18:	FB_FileClose_Indo.bExecute:=TRUE;
	 IF NOT FB_FileClose_Indo.bBusy AND NOT FB_FileClose_Indo.bError THEN
	IndoReport:=20;END_IF

19:	IF bANewDay THEN
	IndoReport:=IndoReport+1;
	ELSIF NOT bANewDay THEN FB_FileOpen_Indo.bExecute:=FALSE; IndoReport:=9;
	END_IF

20:	FB_FileOpen_Indo.bExecute:=FALSE;SerialNo:=SerialNo+1;IndoReport:=9;
END_CASE

	IF sDay <> sOldDay THEN
	bANewDay:=TRUE;IndoReport:=0; SerialNo:=0;END_IF
	TON_NEWDAY(IN:=bANewDay , PT:=T#0.5s , Q=> , ET=> );

CASE WriteError OF

0:	IF FB_FileWrite_Indo.bError THEN
	FB_FileWrite_Indo.bExecute:=FALSE;TON_writedly(IN:=FALSE);
	WriteError:=WriteError+1;END_IF

1:	TON_writedly(IN:=TRUE , PT:=t#2s , Q=> , ET=> );
	IF TON_writedly.Q THEN
	 FB_FileWrite_Indo.bExecute:=TRUE;WriteError:=WriteError+1;END_IF

2:	TON_writedly(IN:=FALSE);WriteError:=0;

END_CASE

CASE OpenError OF

0:	IF FB_FileOpen_Indo.bError THEN
	FB_FileOpen_Indo.bExecute:=FALSE;TON_Opendly(IN:=FALSE);
	OpenError:=OpenError+1;END_IF

1:	TON_Opendly(IN:=TRUE , PT:=t#2s , Q=> , ET=> );
	IF TON_Opendly.Q THEN
	FB_FileOpen_Indo.bExecute:=TRUE;OpenError:=OpenError+1;END_IF

2:	TON_Opendly(IN:=FALSE);OpenError:=0;

END_CASE
END_PROGRAM

(* POU Initialize/Bag_Int, ST *)
PROGRAM Bag_Int
VAR
	BagUnitInt: INT;


END_VAR
CASE BagUnitInt OF

0:	IF bRBagUnitIntRdy  AND NOT bPauseSeq AND NOT bQBagHolder THEN
	bRBagUnitIntRdy:=FALSE;
	BagUnitInt:=BagUnitInt+1;END_IF

1:	IF  bIBagPusherPistonHome THEN BagUnitInt:=BagUnitInt+2;
	ELSIF NOT bIBagPusherPistonHome AND NOT bPauseSeq THEN
	bQRBagPusherForwardPiston:=FALSE;bQRBagPusherReversePiston:= TRUE;END_IF

2:	IF bIBagPusherPistonHome THEN
	bQRBagPusherReversePiston:= FALSE;bQRBagPusherForwardPiston:=FALSE;BagUnitInt:=BagUnitInt+1;END_IF

3:	bRBagUnitIntRdy:=FALSE; BagUnitInt:=BagUnitInt+1;

4:	IF bIBagTiltingPistonHome THEN BagUnitInt:=BagUnitInt+2;
	ELSIF NOT bIBagTiltingPistonHome AND NOT bPauseSeq THEN
	bQRBagTiltingpistonForward:=FALSE;bQRBagTiltingpistonReverse:=TRUE;BagUnitInt:=BagUnitInt+1;END_IF

5:	IF  bIBagTiltingPistonHome THEN
	bQRBagTiltingpistonForward:=FALSE;bQRBagTiltingpistonReverse:=FALSE;BagUnitInt:=BagUnitInt+1;END_IF

6:	bQRColumnStopperPiston:=FALSE;bQRColumnReversePiston:=FALSE;BagUnitInt:=BagUnitInt+1;

7:	IF bISeperatorPlatePistonHome AND bIConePusher1PistonHome AND NOT bQBagHolder
	AND bIBagPusherPistonHome AND bIBagTiltingPistonHome AND NOT bPauseSeq THEN
	bQRBagUp_Down180piston:=TRUE;BagUnitInt:=BagUnitInt+1;END_IF

8:	IF bIBagUpDown180PistonEnd AND NOT bPauseSeq AND NOT bQBagHolder THEN bQRBagUp_Down50piston:=TRUE;BagUnitInt:=BagUnitInt+1;END_IF

9:	IF bIBagUpDown50PistonEnd AND NOT bPauseSeq AND NOT bQBagHolder THEN bQRConePusher1Piston:=TRUE;BagUnitInt:=BagUnitInt+1;END_IF

10:	IF bIConePusher1PistonEnd AND NOT bQBagHolder  AND NOT bPauseSeq THEN bQRConePusher1Piston:=FALSE;BagUnitInt:=BagUnitInt+1;END_IF

11:	IF bISeperatorPlatePistonHome  AND NOT bQBagHolder  AND bIConePusher1PistonHome AND NOT bPauseSeq THEN BagUnitInt:=BagUnitInt+1;END_IF

12:	IF  NOT bPauseSeq AND NOT bQBagHolder  THEN BagUnitInt:=BagUnitInt+1;END_IF

13:	BagUnitInt:=BagUnitInt+1;

14:	BagUnitInt:=BagUnitInt+1;

15:	IF bISeperatorPlatePistonHome AND bIConePusher1PistonHome AND bIBagUpDown50PistonEnd AND bIBagUpDown180PistonEnd
	AND NOT bQBagHolder  AND NOT bPauseSeq THEN
	bQAColumnStopperPiston:=TRUE;
	bQAConePusher3Piston:= TRUE;
	bQABagUp_Down50piston:=TRUE;
	bQABagUp_Down180piston:=TRUE;
	BagUnitInt:=BagUnitInt+1;
	END_IF

16:	IF bIColumnStopperPistonEnd AND bIBagResetPb  THEN IntAllOver:=TRUE;
	bQRBagUp_Down50piston:=FALSE;
	bQRBagUp_Down180piston:=FALSE;
	BagUnitInt:=0;
	END_IF

END_CASE
IF bQRConePusher1Piston AND bIConePusher1SaftyObjectSensor THEN
bAConePusher1SafetyError:=TRUE;bAConePusher1SafetyErrorStatus:='Check Cone Pusher 1';END_IF
IF bErrorReset AND NOT bIConePusher1SaftyObjectSensor THEN
 bAConePusher1SafetyError:=FALSE;bQRConePusher1Piston:=TRUE;bAConePusher1SafetyErrorStatus:='Continue Machine Operation';END_IF

IF bMcStopEnable1 OR NOT bAutoModeOn  THEN
bQRBagUp_Down50piston:=FALSE;
bQRBagUp_Down180piston:=FALSE;
bQABagUp_Down50piston:=FALSE;
bQABagUp_Down180piston:=FALSE;
bQAConePusher3Piston:= FALSE;
bQAColumnStopperPiston:=FALSE;
bQRConePusher1Piston:=FALSE;
bQAConePusher1Piston:=FALSE;
bQRBagTiltingpistonForward:=FALSE;
bQRBagTiltingpistonReverse:=FALSE;
bQRBagPusherForwardPiston:= FALSE;
bQRBagPusherReversePiston:=FALSE;
bQRColumnStopperPiston:=FALSE;
bQRColumnReversePiston:=FALSE;
BagUnitInt:=0;
END_IF
END_PROGRAM

(* POU Initialize/ConeFeedCon_Int, ST *)
PROGRAM ConeFeedCon_Int
VAR

	ConeFeedCon: INT;
	bQRConeFeedCon: BOOL;
	bRConePresentInConeFeedCon: BOOL;
	TON_ConeFeedConInt: TON;
	ConeFeedConIntRunning: BOOL;
	sConeFeedConStatus: STRING;
	ConeFeedConIntOver: BOOL;
END_VAR
CASE ConeFeedCon OF

0: IF bAInitializeSeq AND bPauseSeq AND bAutoModeOn THEN
	ConeFeedCon:=ConeFeedCon+1;END_IF

1:	bQRConeFeedCon:=TRUE;ConeFeedCon:=ConeFeedCon+1;

2:	IF bRConePresentInConeFeedCon THEN
		ConeFeedCon:=ConeFeedCon+2;
		ELSIF NOT bRConePresentInConeFeedCon THEN
		ConeFeedCon:=ConeFeedCon+1;
		END_IF

3:	IF  ConeFeedConIntRunning  AND bRConePresentInConeFeedCon THEN
			ConeFeedCon:=ConeFeedCon+1;
	ELSIF TON_ConeFeedConInt.Q  AND NOT bRConePresentInConeFeedCon THEN
		ConeFeedCon:=ConeFeedCon+3;
	END_IF

4:	bQRConeFeedCon:=FALSE;
	TON_ConeFeedConInt(IN:=FALSE);
	ConeFeedCon:=ConeFeedCon+1;

5:	IF NOT bRConePresentInConeFeedCon AND NOT  bPauseSeq THEN
	ConeFeedCon:=1;END_IF

6:	bQRConeFeedCon:=FALSE;
	TON_ConeFeedConInt(IN:=FALSE);
	ConeFeedCon:=ConeFeedCon+1;

7:	ConeFeedConIntOver:=TRUE;
	ConeFeedCon:=ConeFeedCon+1;

8:	ConeFeedCon:=0;

END_CASE

TON_ConeFeedConInt(IN:=bQRConeFeedCon , PT:=T#10s , Q=> , ET=> );

IF TON_ConeFeedConInt.ET >t#1ms AND  TON_ConeFeedConInt.ET<=t#10s THEN
ConeFeedConIntRunning:=TRUE;
ELSE
ConeFeedConIntRunning:=FALSE;
END_IF


IF (bIConeOrientationTopLimitSwitch OR bIUnit_A_ConeCrossLimitSwitch OR bIUnit_B_ConeCrossLimitSwitch)  AND ConeFeedConIntRunning  THEN
bRConePresentInConeFeedCon:=TRUE;
END_IF

IF  bRConePresentInConeFeedCon AND NOT bIConeOrientationTopLimitSwitch AND NOT  bIUnit_A_ConeCrossLimitSwitch
AND NOT  bIUnit_B_ConeCrossLimitSwitch AND bErrorReset THEN bRConePresentInConeFeedCon:=FALSE;END_IF

IF bRConePresentInConeFeedCon THEN
sConeFeedConStatus:='Clear Cone At Cone Feed Conveyor';
ELSE
sConeFeedConStatus:=' Continue Machine Running ';
END_IF

IF bMcStopEnable1 OR NOT bAutoModeOn  THEN
ConeFeedConIntOver:=FALSE;
ConeFeedConIntRunning:=FALSE;
sConeFeedConStatus:=' Continue Machine Running ';
bRConePresentInConeFeedCon:=FALSE;
bQRConeFeedCon:=FALSE;
bAIntHomeCheckError:=FALSE;
IntAllOver:=FALSE;
bAMachineOn:=FALSE;
bAInitializeSeq:=FALSE;
ConeFeedCon:=0;
END_IF
END_PROGRAM

(* POU Initialize/ConeTransfer_Int, ST *)
PROGRAM ConeTransfer_Int
VAR
	ConeTransferInt: INT;

END_VAR
CASE ConeTransferInt OF

0:	IF TiltIntRdy AND NOT bPauseSeq THEN
	ConeTransferInt:=ConeTransferInt+1;END_IF

1:	IF (bITiltingHome OR bITiltingEnd) AND NOT bPauseSeq THEN
	TiltIntRdy:=FALSE;bQRForwardPiston:=TRUE;bQRReversePiston:=TRUE;ConeTransferInt:=ConeTransferInt+1;END_IF

2:	IF bIForwardPistonEnd AND bIReversePistonEnd AND NOT bPauseSeq AND (bITiltingHome OR bITiltingEnd) THEN
	bQRForwardPiston:=FALSE;bQRReversePiston:=FALSE;ConeTransferInt:=ConeTransferInt+1;END_IF

3:	IF bIForwardPistonHome AND bIReversePistonHome AND NOT bPauseSeq THEN
	ConeTransferInt:=ConeTransferInt+1;END_IF

4:	bHMI_Cone_Tilting_Piston_On:=FALSE;
	bQRTiltingPiston:=FALSE;
	bQATiltingPiston:=FALSE;
	bQM_Cone_Tilting_Piston:=FALSE;
	bQM_Cone_Tilting_Piston_Rev:=TRUE;
	ConeTransferInt:=ConeTransferInt+1;

5:	IF bITiltingHome AND NOT bPauseSeq THEN
	bQM_Cone_Tilting_Piston_Rev:=FALSE;TiltingIntOvr:=TRUE;ConeTransferInt:=ConeTransferInt+1;END_IF

6:	ConeTransferInt:=0;

END_CASE

IF bMcStopEnable1 OR NOT bAutoModeOn  THEN
TiltingIntOvr:=FALSE;bQRForwardPiston:=FALSE;bQRReversePiston:=FALSE;ConeTransferInt:=0;END_IF
END_PROGRAM

(* POU Initialize/Main_Int, ST *)
PROGRAM Main_Int
VAR
	R_TRIG_1: R_TRIG;
END_VAR
(*************************    INITIAL ERROR CHECK*************************)
IF bMCStartInAuto AND bAutoModeOn   AND NOT bASupplyPressureError
 AND NOT bMcStopEnable AND (bABagModeSelected OR bABoxModeSelected)
	AND NOT IntAllOver  AND NOT bAMainIntStarted THEN  bAMachineOn:=TRUE;END_IF

IF bAInitializeSeq OR bMcStopEnable THEN   bAMachineOn:=FALSE;END_IF

(*IF bAMachineOn AND NOT bIUnit_A_RowStopperHome THEN bAError1:=TRUE;bAError1Status:='Check Row Stopper A Home';END_IF
IF bAMachineOn AND NOT bIUnit_B_RowStopperHome THEN bAError2:=TRUE;bAError2Status:='Check Row Stopper B Home';END_IF*)
IF bAMachineOn AND NOT bIConeFeedingPistonHome THEN bAError3:=TRUE;bAError3Status:='Check Cone Feed Piston Home';END_IF
IF bAMachineOn AND NOT bIForwardPistonHome THEN bAError4:=TRUE;bAError4Status:='Check Forward Piston Home';END_IF
IF bAMachineOn AND NOT bIReversePistonHome THEN bAError5:=TRUE;bAError5Status:='Check Reverse Piston  Home';END_IF
(*IF bAMachineOn AND NOT bITiltingHome THEN bAError6:=TRUE;bAError6Status:='Check Tilting Home';END_IF*)
IF bAMachineOn AND NOT bIWrappingChanelPiston1Home THEN bAError7:=TRUE;bAError7Status:='Check Wrapping Piston 1  Home';END_IF
IF bAMachineOn AND NOT bIWrappingChanelPiston2Home THEN bAError8:=TRUE;bAError8Status:='Check Wrapping Piston 2 Home';END_IF
IF bAMachineOn AND NOT bISealingTopPistonHome THEN bAError9:=TRUE;bAError9Status:='Check Sealing Top Piston Home';END_IF
IF bAMachineOn AND NOT bISealingBottomPistonHome THEN bAError10:=TRUE;bAError10Status:='Check Sealing Bottom PistonHome';END_IF
IF bAMachineOn AND NOT bISealingSeparatorXAxisPistonHome THEN bAError11:=TRUE;bAError11Status:='Check X Axis Piston Home';END_IF
IF bAMachineOn AND NOT bISealingSeparatorYAxisPistonHome THEN bAError12:=TRUE;bAError12Status:='Check Y Axis Piston Home';END_IF
IF bAMachineOn AND NOT bIColumnStopperPistonHome THEN bAError13:=TRUE;bAError13Status:='Check Column Stopper Home';END_IF
IF bAMachineOn AND NOT bIColumnReversePistonHome THEN bAError14:=TRUE;bAError14Status:='Check Cone Reverse Piston Home';END_IF
IF bAMachineOn AND NOT bISeperatorPlatePistonHome THEN bAError15:=TRUE;bAError15Status:='Check Seperator Piston Home';END_IF
IF bAMachineOn AND NOT bIConePusher1PistonHome THEN bAError16:=TRUE;bAError16Status:='Check Cone Pusher 2 Home';END_IF
IF bAMachineOn AND NOT bIBagUpDown50PistonHome THEN bAError17:=TRUE;bAError17Status:='Check Up Down Piston 50 Home';END_IF
IF bAMachineOn AND NOT bIBagUpDown180PistonHome THEN bAError18:=TRUE;bAError18Status:='Check Up Down Piston 180 Home';END_IF
IF bAMachineOn AND NOT bIBagPusherPistonHome THEN bAError19:=TRUE;bAError19Status:='Check Bag Pusher Home';END_IF
IF bAMachineOn AND NOT bIBagTiltingPistonHome THEN bAError20:=TRUE;bAError20Status:='Check Bag Tilting Home';END_IF

(*IF bErrorReset AND bAMachineOn AND bIUnit_A_RowStopperHome  AND NOT IntAllOver THEN bAError1:=FALSE;bAError1Status:='Continue Machine Running';END_IF

IF bErrorReset AND bAMachineOn AND bIUnit_B_RowStopperHome  AND NOT IntAllOver THEN bAError2:=FALSE;bAError2Status:='Continue Machine Running';END_IF*)

IF bErrorReset AND bAMachineOn AND bIConeFeedingPistonHome  AND NOT IntAllOver THEN bAError3:=FALSE;bAError3Status:='Continue Machine Running';END_IF

IF bErrorReset AND bAMachineOn AND bIForwardPistonHome  AND NOT IntAllOver THEN bAError4:=FALSE;bAError4Status:='Continue Machine Running';END_IF

IF bErrorReset AND bAMachineOn AND bIReversePistonHome  AND NOT IntAllOver THEN bAError5:=FALSE;bAError5Status:='Continue Machine Running';END_IF

(*IF bErrorReset AND bAMachineOn AND bITiltingHome  AND NOT IntAllOver THEN bAError6:=FALSE;bAError6Status:='Continue Machine Running';END_IF*)

IF bErrorReset AND bAMachineOn AND bIWrappingChanelPiston1Home  AND NOT IntAllOver THEN bAError7:=FALSE;bAError7Status:='Continue Machine Running';END_IF

IF bErrorReset AND bAMachineOn AND bIWrappingChanelPiston2Home  AND NOT IntAllOver THEN bAError8:=FALSE;bAError8Status:='Continue Machine Running';END_IF

IF bErrorReset AND bAMachineOn AND bISealingTopPistonHome  AND NOT IntAllOver THEN bAError9:=FALSE;bAError9Status:='Continue Machine Running';END_IF

IF bErrorReset AND bAMachineOn AND bISealingBottomPistonHome  AND NOT IntAllOver THEN bAError10:=FALSE;bAError10Status:='Continue Machine Running';END_IF

IF bErrorReset AND bAMachineOn AND bISealingSeparatorXAxisPistonHome  AND NOT IntAllOver THEN bAError11:=FALSE;bAError11Status:='Continue Machine Running';END_IF

IF bErrorReset AND bAMachineOn AND bISealingSeparatorYAxisPistonHome   AND NOT IntAllOver THEN bAError12:=FALSE;bAError12Status:='Continue Machine Running';END_IF

IF bErrorReset AND bAMachineOn AND bIColumnStopperPistonHome  AND NOT IntAllOver THEN bAError13:=FALSE;bAError13Status:='Continue Machine Running';END_IF

IF bErrorReset AND bAMachineOn AND bIColumnReversePistonHome  AND NOT IntAllOver THEN bAError14:=FALSE;bAError14Status:='Continue Machine Running';END_IF

IF bErrorReset AND bAMachineOn AND bISeperatorPlatePistonHome  AND NOT IntAllOver THEN bAError15:=FALSE;bAError15Status:='Continue Machine Running';END_IF

IF bErrorReset AND bAMachineOn AND bIConePusher1PistonHome  AND NOT IntAllOver THEN bAError16:=FALSE;bAError16Status:='Continue Machine Running';END_IF

IF bErrorReset AND bAMachineOn AND bIBagUpDown50PistonHome  AND NOT IntAllOver THEN bAError17:=FALSE;bAError17Status:='Continue Machine Running';END_IF

IF bErrorReset AND bAMachineOn AND bIBagUpDown180PistonHome  AND NOT IntAllOver THEN bAError18:=FALSE;bAError18Status:='Continue Machine Running';END_IF

IF bErrorReset AND bAMachineOn AND bIBagPusherPistonHome  AND NOT IntAllOver THEN bAError19:=FALSE;bAError19Status:='Continue Machine Running';END_IF

IF bErrorReset AND bAMachineOn AND bIBagTiltingPistonHome  AND NOT IntAllOver THEN bAError20:=FALSE;bAError20Status:='Continue Machine Running';END_IF

IF bAError1 OR bAError2 OR bAError3 OR bAError4 OR bAError5 OR bAError6 OR bAError7 OR bAError8 OR bAError9 OR bAError10 OR
bAError11 OR bAError12 OR bAError13 OR bAError14 OR bAError15 OR bAError16 OR bAError17 OR bAError18 OR bAError19 OR bAError20 THEN
bAIntHomeCheckError:=TRUE;
ELSE bAIntHomeCheckError:=FALSE;END_IF
										(***MAIN INT***)
IF Initialize_TapHmi  AND bMcStartInAuto AND bAutoModeOn AND NOT bASupplyPressureError
	 AND (bABagModeSelected OR bABoxModeSelected) AND NOT bAIntHomeCheckError
	AND NOT IntAllOver AND NOT  bMcStopEnable AND NOT bAMainIntStarted THEN
	bAInitializeSeq:=TRUE;
	bAMainIntStarted:=TRUE;
ELSE
	bAInitializeSeq:=FALSE;
END_IF


	R_TRIG_1(CLK:= IntAllOver  , Q=> );
IF  bMcStopEnable OR R_TRIG_1.Q   OR NOT bAutoModeOn  THEN bAMainIntStarted:=FALSE; END_IF

IF bMcStopEnable1 OR NOT bAutoModeOn  THEN
bAError1:=FALSE;bAError2:=FALSE;bAError3:=FALSE;bAError4:=FALSE;bAError5:=FALSE;bAError6:=FALSE;bAError7:=FALSE;bAError8:=FALSE;bAError9:=FALSE;bAError10:=FALSE;
bAError11:=FALSE;bAError12:=FALSE;bAError13:=FALSE;bAError14:=FALSE;bAError15:=FALSE;bAError16:=FALSE;bAError17:=FALSE;bAError18:=FALSE;bAError19:=FALSE;bAError20:=FALSE;
bAError1Status:='Continue Machine Running';bAError2Status:='Continue Machine Running';bAError3Status:='Continue Machine Running';bAError4Status:='Continue Machine Running';bAError5Status:='Continue Machine Running';
bAError6Status:='Continue Machine Running';bAError7Status:='Continue Machine Running';bAError8Status:='Continue Machine Running';bAError9Status:='Continue Machine Running';bAError10Status:='Continue Machine Running';
bAError11Status:='Continue Machine Running';bAError12Status:='Continue Machine Running';bAError13Status:='Continue Machine Running';bAError14Status:='Continue Machine Running';bAError15Status:='Continue Machine Running';
bAError16Status:='Continue Machine Running';bAError17Status:='Continue Machine Running';bAError18Status:='Continue Machine Running';bAError19Status:='Continue Machine Running';bAError20Status:='Continue Machine Running';END_IF
END_PROGRAM

(* POU Initialize/Ret_Int, ST *)
PROGRAM Ret_Int
VAR
	Ret_A_Int: INT;
	bQRRetA_RowStopperMotorRev: BOOL;
	Ret_B_Int: INT;
	bQRRetB_RowStopperMotorRev: BOOL;
END_VAR
					(*********************Ret-A Int Logic****************)
CASE Ret_A_Int OF

0:IF bIMcStartPb AND NOT bAMainIntStarted THEN
	Ret_A_Int:=Ret_A_Int+1;END_IF

1:IF bIUnit_A_RowStopperHome THEN Ret_A_Int:=Ret_A_Int+2;
	ELSIF NOT bIUnit_A_RowStopperHome THEN Ret_A_Int:=Ret_A_Int+1;END_IF

2:bQRRetA_RowStopperMotorRev:=TRUE;Ret_A_Int:=Ret_A_Int+1;

3:IF bIUnit_A_RowStopperHome THEN
	bQRRetA_RowStopperMotorRev:=FALSE;Ret_A_Int:=Ret_A_Int+1;END_IF

4:Ret_A_Int:=0;

END_CASE


					(*********************Ret-B Int Logic****************)
CASE Ret_B_Int OF

0:IF bIMcStartPb AND NOT bAMainIntStarted THEN
	Ret_B_Int:=Ret_B_Int+1;END_IF

1:IF bIUnit_B_RowStopperHome THEN Ret_B_Int:=Ret_B_Int+2;
	ELSIF NOT bIUnit_B_RowStopperHome THEN Ret_B_Int:=Ret_B_Int+1;END_IF

2:bQRRetB_RowStopperMotorRev:=TRUE;Ret_B_Int:=Ret_B_Int+1;

3:IF bIUnit_B_RowStopperHome THEN
	bQRRetB_RowStopperMotorRev:=FALSE;Ret_B_Int:=Ret_B_Int+1;END_IF

4:Ret_B_Int:=0;

END_CASE


IF bMcStopEnable1 OR NOT bAutoModeOn  THEN
Ret_A_Int:=0;
Ret_B_Int:=0;
bQRRetA_RowStopperMotorRev:=FALSE;
bQRRetB_RowStopperMotorRev:=FALSE;
END_IF
END_PROGRAM

(* POU Initialize/Sealing_Int, ST *)
PROGRAM Sealing_Int
VAR
	SealConInt:INT;
	TON_SealingConInt:TON;
	SealingPistonInt:INT;
	BagIntCheck:INT;
	TON_SealingPis:TON;
	TON_SealingDly_Int:TON;


END_VAR
CASE SealConInt OF

0:IF (bAInitializeSeq OR bRSealUnitIntOver) AND NOT bPauseSeq AND bAutoModeOn THEN
	SealConInt:=SealConInt+1;END_IF

1:IF WrappingSafety AND NOT bPauseSeq THEN
	bQRSealingConveyorMotor:=TRUE;WrapUnitIntOver:=FALSE;SealConInt:=SealConInt+1;END_IF

2:	IF bRConePresentInSealCon THEN
		SealConInt:=SealConInt+2;
		ELSIF NOT bRConePresentInSealCon THEN
		SealConInt:=SealConInt+1;
		END_IF

3:IF  SealingConIntRunning  AND bRConePresentInSealCon THEN
			SealConInt:=SealConInt+1;
	ELSIF TON_SealingConInt.Q  AND NOT bRConePresentInSealCon THEN
		SealConInt:=SealConInt+3;
	END_IF

4:	bQRSealingConveyorMotor:=FALSE;
	TON_SealingConInt(IN:=FALSE);
	SealConInt:=SealConInt+1;

5:	IF NOT bRConePresentInSealCon AND NOT  bPauseSeq THEN
	SealConInt:=1;END_IF

6:	bQRSealingConveyorMotor:=FALSE;
	TON_SealingConInt(IN:=FALSE);
	SealConInt:=SealConInt+1;

7:	IF bRSealUnitIntOver THEN SealConIntOver:=TRUE;bRSealUnitIntOver:=FALSE;SealConInt:=SealConInt+1;
	ELSIF NOT bRSealUnitIntOver THEN
	SealConInt:=SealConInt+1;END_IF

8:	SealConInt:=0;

END_CASE


TON_SealingConInt(IN:=bQRSealingConveyorMotor , PT:=T#10s , Q=> , ET=> );

IF TON_SealingConInt.ET >t#1ms AND  TON_SealingConInt.ET<=t#10s THEN
SealingConIntRunning:=TRUE;
ELSE
SealingConIntRunning:=FALSE;
END_IF


IF bIConeCountsensor  AND SealingConIntRunning  THEN
bRConePresentInSealCon:=TRUE;
END_IF

IF  bRConePresentInSealCon AND NOT bIConeCountsensor
AND bErrorReset THEN bRConePresentInSealCon:=FALSE;END_IF

IF bRConePresentInSealCon THEN
sSealingConStatus:='Clear Cone At Sealing Conveyor';
ELSE
sSealingConStatus:=' Continue Machine Running ';
END_IF

CASE SealingPistonInt OF

0:	IF WrapUnitIntOver AND WrappingSafety AND NOT bPauseSeq AND bAutoModeOn THEN WrapUnitIntOver:=FALSE;
	bQRSealingSeparatorYAxisPiston:=TRUE;SealingPistonInt:=SealingPistonInt+1;END_IF

1:	IF bISealingSeparatorYAxisPistoEnd AND NOT bPauseSeq THEN SealConIntOver:=FALSE;
	bQRSealingTopPiston:=TRUE;bQRSealingBottomPiston:=TRUE;SealingPistonInt:=SealingPistonInt+1;END_IF

2:	TON_SealingPis(IN:=TRUE , PT:=t#2s , Q=> , ET=> );
	IF (bISealingTopPistonEnd AND bISealingBottomPistonEnd) OR TON_SealingPis.Q THEN
	SealingPistonInt:=SealingPistonInt+1;END_IF

3:	TON_SealingDly_Int(IN:=TRUE , PT:= t#2s, Q=> , ET=> );
	IF TON_SealingDly_Int.Q THEN SealingPistonInt:=SealingPistonInt+1;END_IF

4:	bQRSealingSeparatorXAxisPiston:=TRUE;TON_SealingPis(IN:=FALSE);TON_SealingDly_Int(IN:=FALSE);
	SealingPistonInt:=SealingPistonInt+1;

5:	IF bISealingSeparatorXAxisPistonEnd AND NOT bPauseSeq THEN
	bQRSealingSeparatorYAxisPiston:=FALSE;
	bQRSealingTopPiston:=FALSE;bQRSealingBottomPiston:=FALSE;
	bQRSealingSeparatorXAxisPiston:=FALSE;SealingPistonInt:=SealingPistonInt+1;END_IF

6:	IF SealingSafety AND NOT bPauseSeq THEN
	bRSealUnitIntOver:=TRUE;SealingPistonInt:=SealingPistonInt+1;END_IF

7:	SealingPistonInt:=0;

END_CASE

CASE BagIntCheck OF

0: 	IF bABagModeSelected AND NOT bPauseSeq AND SealConIntOver  THEN
	bRBagUnitIntRdy:=TRUE;SealConIntOver:=FALSE;
	ELSIF bABoxModeSelected AND NOT bPauseSeq AND SealConIntOver  THEN
	IntAllOver:=TRUE;SealConIntOver:=FALSE; TiltingIntOvr:=FALSE;BagIntCheck:=BagIntCheck+1;END_IF

1:	BagIntCheck:=0;
END_CASE;


IF bMcStopEnable1 OR NOT bAutoModeOn  THEN
bRSealUnitIntOver:=FALSE;SealingPistonInt:=0;bQRSealingSeparatorYAxisPiston:=FALSE;
	bQRSealingTopPiston:=FALSE;bQRSealingBottomPiston:=FALSE;
	bQRSealingSeparatorXAxisPiston:=FALSE;TON_SealingDly_Int(IN:=FALSE);SealConIntOver:=FALSE;
TON_SealingPis(IN:=FALSE);SealConIntOver:=FALSE;SealingConIntRunning:=FALSE;
bRConePresentInSealCon:=FALSE;TON_SealingConInt(IN:=FALSE);
bQRSealingConveyorMotor:=FALSE;WrapUnitIntOver:=FALSE;SealConInt:=0;BagIntCheck:=0;
END_IF
END_PROGRAM

(* POU Initialize/Wrapping_Int, ST *)
PROGRAM Wrapping_Int
VAR
	WrapConInt: INT;

	TON_WrappingConInt: TON;
	WrapPistonInt: INT;


END_VAR
CASE WrapConInt OF

0:IF (bAInitializeSeq OR TiltingIntOvr ) AND NOT bPauseSeq AND bAutoModeOn THEN
	WrapConInt:=WrapConInt+1;END_IF

1:IF WrappingSafety AND NOT bPauseSeq THEN
	bQRWappingConveyorMotor:=TRUE;WrapConInt:=WrapConInt+1;END_IF

2:	IF bRConePresentInWrapCon THEN
		WrapConInt:=WrapConInt+2;
		ELSIF NOT bRConePresentInWrapCon THEN
		WrapConInt:=WrapConInt+1;
		END_IF

3:IF  WrappingConIntRunning  AND bRConePresentInWrapCon THEN
			WrapConInt:=WrapConInt+1;
	ELSIF TON_WrappingConInt.Q  AND NOT bRConePresentInWrapCon THEN
		WrapConInt:=WrapConInt+3;
	END_IF

4:	bQRWappingConveyorMotor:=FALSE;
	TON_WrappingConInt(IN:=FALSE);
	WrapConInt:=WrapConInt+1;

5:	IF NOT bRConePresentInWrapCon AND NOT  bPauseSeq THEN
	WrapConInt:=1;END_IF

6:	bQRWappingConveyorMotor:=FALSE;
	TON_WrappingConInt(IN:=FALSE);
	WrapConInt:=WrapConInt+1;

7:	IF TiltingIntOvr THEN WrapConIntOver:=TRUE;TiltingIntOvr:=FALSE;WrapConInt:=WrapConInt+1;
	ELSIF NOT TiltingIntOvr THEN
	TiltIntRdy:=TRUE;
	WrapConInt:=WrapConInt+1;END_IF

8:	WrapConInt:=0;

END_CASE


TON_WrappingConInt(IN:=bQRWappingConveyorMotor , PT:=T#10s , Q=> , ET=> );

IF TON_WrappingConInt.ET >t#1ms AND  TON_WrappingConInt.ET<=t#10s THEN
WrappingConIntRunning:=TRUE;
ELSE
WrappingConIntRunning:=FALSE;
END_IF


IF (bIWrappingCone1 OR bIWrappingCone2)  AND WrappingConIntRunning  THEN
bRConePresentInWrapCon:=TRUE;
END_IF

IF  bRConePresentInWrapCon AND NOT bIWrappingCone1 AND NOT  bIWrappingCone2
AND bErrorReset THEN bRConePresentInWrapCon:=FALSE;END_IF

IF bRConePresentInWrapCon THEN
sWrappingConStatus:='Clear Cone At Wrapping Conveyor';
END_IF

CASE WrapPistonInt OF

0:	IF WrapConIntOver AND NOT bPauseSeq AND SealingSafety THEN
	bQRWrappingPiston1:=TRUE;bQRWrappingPiston2:=TRUE;WrapConIntOver:=FALSE;WrapPistonInt:=WrapPistonInt+1;END_IF

1:	 IF NOT bPauseSeq AND NOT bAWrappingPiston1RsError AND NOT bAWrappingPiston2RsError AND
	bIWrappingChanelPiston1End AND bIWrappingChanelPiston2End THEN
	bQRWrappingPiston1:=FALSE;bQRWrappingPiston2:=FALSE;WrapPistonInt:=WrapPistonInt+1;END_IF

2:	 IF  NOT bPauseSeq AND WrappingSafety THEN
	WrapUnitIntOver:=TRUE;WrapPistonInt:=WrapPistonInt+1;END_IF

3:	WrapPistonInt:=0;

END_CASE


IF bMcStopEnable1 OR NOT bAutoModeOn  THEN
WrapPistonInt:=0;WrapConIntOver:=FALSE;bAWrappingPiston1RsError:=FALSE;bAWrappingPiston2RsError:=FALSE;
bQRWrappingPiston1:=FALSE;bQRWrappingPiston2:=FALSE;WrapUnitIntOver:=FALSE;
WrappingConIntRunning:=FALSE;bRConePresentInWrapCon:=FALSE;WrapConInt:=0;TON_WrappingConInt(IN:=FALSE);
bQRWappingConveyorMotor:=FALSE;END_IF
END_PROGRAM

(* POU Manual, ST *)
PROGRAM Manual
VAR

	step: INT;
	Timer1: TON;


END_VAR
					(*************SEALING SAFETY*********************)

IF	bISealingTopPistonHome AND bISealingBottomPistonHome AND bISealingSeparatorYAxisPistonHome AND bISealingSeparatorXAxisPistonHome
THEN
	SealingSafety:=TRUE;
ELSE
	SealingSafety:=FALSE;
END_IF

						(*************WRAPPING  SAFETY*********************)
IF 	bIWrappingChanelPiston1Home AND  bIWrappingChanelPiston2Home
THEN
	WrappingSafety:=TRUE;
ELSE
	WrappingSafety:=FALSE;
END_IF

					(*======================MANUAL SEALING LOGIC==========================*)

IF NOT  bAutoModeOn AND bIManualSealingPb THEN
	bManualSealEnable:=TRUE;
ELSE bManualSealEnable:=FALSE; END_IF

IF   bAutoModeOn AND bPauseSeq  AND bIManualSealingPb THEN
bManualSealEnable2:=TRUE;
ELSE bManualSealEnable2:=FALSE; END_IF

CASE step OF

	0:	IF  ( bManualSealEnable OR bManualSealEnable2  )THEN bMManualSealOn:=TRUE; step:=step+1;  END_IF

	1:	Timer1(IN:= FALSE);
		bQM_Cone_Sealing_Bottom_Piston:=TRUE;
		bQM_Cone_Sealing_Top_Piston:=TRUE;
		step:=step+1;

	2:	 IF bISealingBottomPistonEnd AND bISealingTopPistonEnd THEN
		 step:=step+1;
		END_IF

	3:	Timer1(IN:=TRUE , PT:=t#3s , Q=> , ET=> );
		IF Timer1.Q THEN step:=step+1; END_IF

	4:	bMManualSealOn:=FALSE;
		bQM_Cone_Sealing_Bottom_Piston:=FALSE;
		bQM_Cone_Sealing_Top_Piston:=FALSE;
		Timer1(IN:= FALSE);
		 step:=step+1;

	5:	step:=0;
END_CASE

								(*************RET-A FWD ; REV *********************)
IF bHMI_RetA_Fwd_On AND NOT bHMI_RetA_Rev_On AND NOT  bQM_RetA_Rev THEN bQM_RetA_Fwd:=TRUE;ELSE bQM_RetA_Fwd:=FALSE;END_IF

IF bHMI_Ret_RevA_On AND NOT bHMI_RetA_Fwd_On AND NOT bQM_RetA_Fwd THEN bQM_RetA_Rev:=TRUE;ELSE bQM_RetA_Rev:=FALSE;END_IF

bQMRetA_RowStopperMotorFwd:=bQM_RetA_Fwd;
bQMRetA_RowStopperMotorRev:=bQM_RetA_Rev;

								(*************RET-A FWD ; REV *********************)
IF bHMI_RetB_Fwd_On AND NOT bHMI_RetB_Rev_On AND NOT  bQM_RetB_Rev THEN bQM_RetB_Fwd:=TRUE;ELSE bQM_RetB_Fwd:=FALSE;END_IF

IF bHMI_Ret_RevB_On AND NOT bHMI_RetB_Fwd_On AND NOT bQM_RetB_Fwd THEN bQM_RetB_Rev:=TRUE;ELSE bQM_RetB_Rev:=FALSE;END_IF

bQMRetB_RowStopperMotorFwd:=bQM_RetB_Fwd;
bQMRetB_RowStopperMotorRev:=bQM_RetB_Rev;


								(*************CONE FEEDING PISTON*********************)
IF bHMI_Cone_Feeding_Piston_On THEN
	bQM_Cone_Feeding_Piston:=TRUE;
ELSE bQM_Cone_Feeding_Piston:=FALSE;END_IF
bQMConeFeedingPiston:=bQM_Cone_Feeding_Piston;

								(*************CONE FORWARD PISTON*********************)
IF bHMI_Cone_Forward_Piston_On AND (bITiltingHome OR bITiltingEnd) THEN
bQM_Cone_Forward_Piston:=TRUE;
ELSE bQM_Cone_Forward_Piston:=FALSE;END_IF
bQMForwardPiston:=bQM_Cone_Forward_Piston;

								(*************CONE REVERSE PISTON*********************)
IF bHMI_Cone_Reverse_Piston_On AND (bITiltingHome OR bITiltingEnd) THEN
bQM_Cone_Reverse_Piston:=TRUE;
ELSE bQM_Cone_Reverse_Piston:=FALSE;END_IF
bQMReversePiston:=bQM_Cone_Reverse_Piston;

								(*************CONE TILTING PISTON*********************)
IF bHMI_Cone_Tilting_Piston_On AND bIForwardPistonHome AND bIReversePistonHome THEN
bQM_Cone_Tilting_Piston:=TRUE;bQM_Cone_Tilting_Piston_Rev:=FALSE; END_IF
IF NOT bHMI_Cone_Tilting_Piston_On THEN bQM_Cone_Tilting_Piston:=FALSE;END_IF;
bQMTiltingPiston:=bQM_Cone_Tilting_Piston;

								(*************WRAPPING PISTON 1*********************)
IF bHMI_Cone_Wrapping_Piston1_On AND SealingSafety THEN
bQM_Cone_Wrapping_Piston1_Rev:=FALSE;bQM_Cone_Wrapping_Piston1_Fwd:=TRUE;
ELSE bQM_Cone_Wrapping_Piston1_Fwd:=FALSE;END_IF
bQMWrappingPiston1:=bQM_Cone_Wrapping_Piston1_Fwd;

IF bHMI_Cone_Wrapping_Piston1_On_Rev AND SealingSafety THEN
bQM_Cone_Wrapping_Piston1_Fwd:=FALSE;bQM_Cone_Wrapping_Piston1_Rev:=TRUE;
ELSE bQM_Cone_Wrapping_Piston1_Rev:=FALSE;END_IF

					(*************WRAPPING PISTON 2*********************)
IF bHMI_Cone_Wrapping_Piston2_On AND SealingSafety THEN
bQM_Cone_Wrapping_Piston2_Rev:=FALSE;bQM_Cone_Wrapping_Piston2_Fwd:=TRUE;
ELSE bQM_Cone_Wrapping_Piston2_Fwd:=FALSE;END_IF
bQMWrappingPiston2:=bQM_Cone_Wrapping_Piston2_Fwd;

IF bHMI_Cone_Wrapping_Piston2_On_Rev AND SealingSafety THEN
bQM_Cone_Wrapping_Piston2_Fwd:=FALSE;bQM_Cone_Wrapping_Piston2_Rev:=TRUE;
ELSE bQM_Cone_Wrapping_Piston2_Rev:=FALSE;END_IF


								(*************SEALING TOP PISTON*********************)
IF bHMI_Cone_Sealing_Top_Piston_On AND WrappingSafety THEN
bQM_Cone_Sealing_Top_Piston:=TRUE;ELSE bQM_Cone_Sealing_Top_Piston:=FALSE;END_IF
bQMSealingTopPiston:=bQM_Cone_Sealing_Top_Piston;


								(*************SEALING BOTTOM PISTON*********************)
IF bHMI_Cone_Sealing_Bottom_Piston_On AND WrappingSafety THEN
bQM_Cone_Sealing_Bottom_Piston:=TRUE;
ELSE bQM_Cone_Sealing_Bottom_Piston:=FALSE;END_IF
bQMSealingBottomPiston:=bQM_Cone_Sealing_Bottom_Piston;


								(*************SEALING Y AXIS  PISTON*********************)
IF bHMI_Cone_Sealing_YAxis_Piston_On AND WrappingSafety THEN
bQM_Cone_Sealing_YAxis_Piston:=TRUE;ELSE bQM_Cone_Sealing_YAxis_Piston:=FALSE;END_IF
bQMSealingSeparatorYAxisPiston:=bQM_Cone_Sealing_YAxis_Piston;


								(*************SEALING X AXIS  PISTON*********************)
IF bHMI_Cone_Sealing_XAxis_Piston_On AND WrappingSafety THEN
bQM_Cone_Sealing_XAxis_Piston:=TRUE;ELSE bQM_Cone_Sealing_XAxis_Piston:=FALSE;END_IF
bQMSealingSeparatorXAxisPiston:=bQM_Cone_Sealing_XAxis_Piston;

								(*************CONE COUNT  PISTON*********************)
IF bHMI_Cone_Count_Piston_On  THEN
bQM_Cone_Count_Piston:=TRUE;ELSE bQM_Cone_Count_Piston:=FALSE;END_IF
bQMConeCountPiston:=bQM_Cone_Count_Piston;

								(*************CONE FEEDING CONVEYOR MOTOR*********************)
IF bHMI_Cone_Feeding_Conveyor_On THEN
bQM_Cone_Feeding_Conveyor:=TRUE;
ELSE bQM_Cone_Feeding_Conveyor:=FALSE;END_IF
bQMFeedingConveyorMotor:=bQM_Cone_Feeding_Conveyor;


								(*************CONE WRAPPING CONVEYOR MOTOR*********************)
IF bHMI_Cone_Wrapping_Conveyor_On THEN
bQM_Cone_Wrapping_Conveyor:=TRUE;ELSE bQM_Cone_Wrapping_Conveyor:=FALSE;END_IF
bQMWappingConveyorMotor:=bQM_Cone_Wrapping_Conveyor;


								(*************CONE SEALING CONVEYOR MOTOR*********************)
IF bHMI_Cone_Sealing_Conveyor_On THEN
bQM_Cone_Sealing_Conveyor:=TRUE;
ELSE bQM_Cone_Sealing_Conveyor:=FALSE;END_IF
bQMSealingConveyorMotor:=bQM_Cone_Sealing_Conveyor;



										(***CONE PUSHER 1***)
IF bIConePusher1_On_Hmi THEN
bQMConePusher1:=TRUE;
ELSE bQMConePusher1:=FALSE;END_IF
bQMSeparatorplatePiston:=bQMConePusher1;


										(***CONE PUSHER 2***)
IF bIConePusher2_On_Hmi THEN
bQMConePusher2:=TRUE;ELSE
bQMConePusher2:=FALSE;END_IF
bQMConePusher1Piston:=bQMConePusher2;


										(***CONE PUSHER 3***)
IF bIConePusher3_On_Hmi THEN
bQMConePusher3:=TRUE;
ELSE bQMConePusher3:=FALSE;END_IF
bQMConePusher2Piston:=bQMConePusher3;


										(***BAG PUSHER FORWARD***)
IF bIBagPusherFwd_On_Hmi THEN
bQMBagPusherFwd:=TRUE;
ELSE bQMBagPusherFwd:=FALSE;END_IF
bQMBagPusherForwardPiston:=bQMBagPusherFwd;


										(***BAG PUSHER REVERSE***)
IF bIBagPusherRev_On_Hmi THEN
bQMBagPusherRev:=TRUE;
ELSE bQMBagPusherRev:=FALSE;END_IF
bQMBagPusherReversePiston:=bQMBagPusherRev;


										(***UP DOWN PISTON 1***)
IF bIUpDownPiston_1_On_Hmi THEN
bQMUpDownPiston_1:=TRUE;
ELSE bQMUpDownPiston_1:=FALSE;END_IF
bQMBagUp_Down180piston:=bQMUpDownPiston_1;


										(***UP DOWN PISTON 2***)
IF bIUpDownPiston_2_On_Hmi THEN
bQMUpDownPiston_2:=TRUE;
ELSE bQMUpDownPiston_2:=FALSE;END_IF
bQMBagUp_Down50piston:=bQMUpDownPiston_2;



										(***BAG TILTING FORWARD***)
IF bIBagTiltingFwd_On_Hmi THEN
bQMBagTiltingFwd:=TRUE;
ELSE bQMBagTiltingFwd:=FALSE;END_IF
bQMBagTiltingpistonForward:=bQMBagTiltingFwd;


										(***BAG TILTING REVERSE***)
IF bIBagTiltingRev_On_Hmi THEN
bQMBagTiltingRev:=TRUE;
ELSE bQMBagTiltingRev:=FALSE;END_IF
bQMBagTiltingpistonReverse:=bQMBagTiltingRev;


										(***bQRColumn Stopper Piston ***)
IF bIColumn_Stopper_Piston_On_Hmi THEN
bQMColumnStopperPiston:=TRUE;
ELSE bQMColumnStopperPiston:=FALSE;END_IF
bQMColumnStopperPiston:=bQMColumnStopperPiston;


										(***bQRColumn Stopper Piston ***)
IF bIColumnConeForwardPiston_On_Hmi THEN
bQMColumnConeForwardPiston:=TRUE;
ELSE bQMColumnConeForwardPiston:=FALSE;END_IF
bQMColumnReversePiston:=bQMColumnConeForwardPiston;


																(***BAG HOLDER ***)
IF   (bAutoModeOn    AND (bIBagHolder_On OR bIBagHolder_On_Hmi)
AND bIBagPusherHome) OR (bManualModeOn AND  (bIBagHolder_On OR bIBagHolder_On_Hmi) AND bIBagPusherHome) THEN
bQMBagHolderPiston:=TRUE;
ELSE bQMBagHolderPiston:=FALSE;END_IF

										(***BAG ROW HOLDER ***)
IF bIBagRowHolderPiston_On_Hmi THEN bQMBagRowHolderPiston:=TRUE;
ELSE bQMBagRowHolderPiston:=FALSE;END_IF
bQBagRowHolderpiston:=bQMBagRowHolderPiston;



IF  bIMcStopPb OR  Stop_TapHmi OR NOT bIEmergencySwitchPb OR NOT  bManualModeOn  THEN
	bHMI_RetA_Fwd_On:=FALSE;
	bHMI_RetA_Rev_On:=FALSE;
	bHMI_RetB_Fwd_On:=FALSE;
	bHMI_RetB_Rev_On:=FALSE;
	bHMI_Cone_Feeding_Piston_On  :=FALSE;
	bHMI_Cone_Forward_Piston_On:=FALSE;
	bHMI_Cone_Reverse_Piston_On :=FALSE;
	bHMI_Cone_Wrapping_Piston1_On :=FALSE;
	bHMI_Cone_Wrapping_Piston2_On :=FALSE;
	bHMI_Cone_Sealing_YAxis_Piston_On :=FALSE;
	bHMI_Cone_Sealing_XAxis_Piston_On :=FALSE;
	bHMI_Cone_Sealing_Top_Piston_On :=FALSE;
	bHMI_Cone_Sealing_Bottom_Piston_On :=FALSE;
	bHMI_Cone_Feeding_Conveyor_On :=FALSE;
	bHMI_Cone_Wrapping_Conveyor_On :=FALSE;
	bHMI_Cone_Sealing_Conveyor_On :=FALSE;
	bQM_RetB_Fwd:=FALSE;
	bQM_RetB_Rev:=FALSE;
	bQM_Cone_Feeding_Piston:=FALSE;
	bQM_Cone_Forward_Piston:=FALSE;
	bQM_Cone_Reverse_Piston:=FALSE;
	bQM_Cone_Sealing_YAxis_Piston:=FALSE;
	bQM_Cone_Sealing_XAxis_Piston:=FALSE;
	bQM_Cone_Feeding_Conveyor:=FALSE;
 	bQM_Cone_Wrapping_Conveyor:=FALSE;
	bQM_Cone_Sealing_Conveyor:=FALSE;
	bQMConePusher1:=FALSE;
	bQMConePusher2:=FALSE;
	bQMConePusher3:=FALSE;
	bQMBagPusherFwd:=FALSE;
	bQMBagPusherRev:=FALSE;
	bQMUpDownPiston_1:=FALSE;
	bQMUpDownPiston_2:=FALSE;
	bQMBagTiltingFwd:=FALSE;
	bQMBagTiltingRev:=FALSE;
	bQMColumnStopperPiston:=FALSE;
	bQMColumnConeForwardPiston:=FALSE;
	bQM_RetA_Rev:=FALSE;
	bQM_RetA_Fwd:=FALSE;
	bQM_RetB_Rev:=FALSE;
	bQM_RetB_Fwd:=FALSE;
	bIConePusher1_On_Hmi:=FALSE;
	bIConePusher2_On_Hmi:=FALSE;
	bIConePusher3_On_Hmi:=FALSE;
	bIBagPusherFwd_On_Hmi:=FALSE;
	bIBagPusherRev_On_Hmi:=FALSE;
	bIUpDownPiston_1_On_Hmi:=FALSE;
	bIUpDownPiston_2_On_Hmi:=FALSE;
	bIBagTiltingFwd_On_Hmi:=FALSE;
	bIBagTiltingRev_On_Hmi:=FALSE;
	bIColumn_Stopper_Piston_On_Hmi:=FALSE;
	bIColumnConeForwardPiston_On_Hmi:=FALSE;
	bIBagHolder_On_Hmi:=FALSE;
	bQM_Cone_Sealing_Top_Piston:=FALSE;
	bQM_Cone_Sealing_Bottom_Piston:=FALSE;
	step:=0;
END_IF
END_PROGRAM

(* POU Weight_Read, ST *)
PROGRAM Weight_Read
VAR
	COMportControl_1: SerialLineControl;
	COMin_1_COMPort_1 AT %I*: EL6inData22B;
	COMOut_1_COMPort_1 AT %Q*: EL6outData22B;
	TxBuffer1: ComBuffer;
	RxBuffer1: ComBuffer;
	ipos_1: INT;
	samplestring_1: STRING;
	ReceiveString_sample_1: ReceiveString;
	resultWt_1: STRING;
	COMportControlError_1: BOOL;
	COMportControlErrorID_1: ComError_t;
	Ret_AWt: REAL;


	COMportControl_2: SerialLineControl;
	COMin_2_COMPort_2 AT %I*: EL6inData22B;
	COMOut_2_COMPort_2 AT %Q*: EL6outData22B;
	TxBuffer2: ComBuffer;
	RxBuffer2: ComBuffer;
	ipos_2: INT;
	samplestring_2: STRING;
	ReceiveString_sample_2: ReceiveString;
	resultWt_2: STRING;
	COMportControlError_2: BOOL;
	COMportControlErrorID_2: ComError_t;
	Ret_BWt: REAL;

END_VAR
(*==============Ret - A Weight Read==================*)

COMportControl_1(
	Mode:= SERIALLINEMODE_EL6_22B,
	pComIn:= ADR(COMin_1_COMport_1),
	pComOut:= ADR(COMout_1_COMport_1),
	SizeComIn:= SIZEOF(COMin_1_COMport_1),
	TxBuffer:= TxBuffer1,
	RxBuffer:= RxBuffer1,
	Error=> COMportControlError_1,
	ErrorID=> COMportControlErrorID_1);

ReceiveString_sample_1(
	Prefix:='w' ,
	Suffix:='g' ,
	Timeout:= t#5s,
	Reset:= ,
	ReceivedString:=samplestring_1 ,
	RXbuffer:= RxBuffer1,
	StringReceived=> ,
	Busy=> ,
	Error=> ,
	RxTimeout=> );
ipos_1:=FIND(samplestring_1,'n');

resultWt_1:= MID (samplestring_1,9,ipos_1+1);
Ret_AWt:=STRING_TO_REAL(resultWt_1);


(*==============Ret - B Weight Read==================*)

COMportControl_2(
	Mode:= SERIALLINEMODE_EL6_22B,
	pComIn:= ADR(COMin_2_COMport_2),
	pComOut:= ADR(COMout_2_COMport_2),
	SizeComIn:= SIZEOF(COMin_2_COMport_2),
	TxBuffer:= TxBuffer2,
	RxBuffer:= RxBuffer2,
	Error=> COMportControlError_2,
	ErrorID=> COMportControlErrorID_2);

ReceiveString_sample_2(
	Prefix:='w' ,
	Suffix:='g' ,
	Timeout:= t#5s,
	Reset:= ,
	ReceivedString:=samplestring_2 ,
	RXbuffer:= RxBuffer2,
	StringReceived=> ,
	Busy=> ,
	Error=> ,
	RxTimeout=> );
ipos_1:=FIND(samplestring_2,'n');

resultWt_2:= MID (samplestring_1,9,ipos_2+1);
Ret_BWt:=STRING_TO_REAL(resultWt_2);
END_PROGRAM

(* POU Alarms/Piston_Alarms, ST *)
PROGRAM Piston_Alarms
VAR
	TON_ConeFeedingPistonOff: BOOL;
	F_TRIG_ConeFeedingPiston: F_TRIG;
	bAConeFeedingPistonOff: BOOL;
	RS_ErrorConeFeedPistonHome: Rs_Error;
	RS_ErrorConeFeedPistonEnd: Rs_Error;
	HMIFeedPistonHome: STRING;
	HMIFeedPistonEnd: STRING;
	HMIFeedPiston: STRING;

	TON_ConeForwardPistonOff: BOOL;
	F_TRIG_ConeForwardPiston: F_TRIG;
	bAConeForwardPistonOff: BOOL;
	RS_ErrorConeForwardPistonHome: Rs_Error;
	RS_ErrorConeForwardPistonEnd: Rs_Error;
	HMIForwardPistonHome: STRING;
	HMIForwardPistonEnd: STRING;
	HMIForwardPiston: STRING;

	TON_ConeReversePistonOff: BOOL;
	F_TRIG_ConeReversePiston: F_TRIG;
	bAConeReversePistonOff: BOOL;
	RS_ErrorConeReversePistonHome: Rs_Error;
	RS_ErrorConeReversePistonEnd: Rs_Error;
	HMIReversePistonHome: STRING;
	HMIReversePistonEnd: STRING;
	HMIReversePiston: STRING;

	TON_ConeTiltingPistonOff: BOOL;
	F_TRIG_ConeTiltingPiston: F_TRIG;
	bAConeTiltingPistonOff: BOOL;
	RS_ErrorConeTiltingPistonHome: Rs_Error;
	RS_ErrorConeTiltingPistonEnd: Rs_Error;
	HMITiltingPistonHome: STRING;
	HMITiltingPistonEnd: STRING;
	HMITiltingPiston: STRING;
	bATiltingPisHomeRsError: BOOL;
	bATiltingPisEndRsError: BOOL;

	TON_Wrapping1PistonOff: BOOL;
	F_TRIG_Wrapping1Piston: F_TRIG;
	bAWrapping1PistonOff: BOOL;
	RS_ErrorWrapping1PistonHome: Rs_Error;
	RS_ErrorWrapping1PistonEnd: Rs_Error;
	HMIWrapping1PistonHome: STRING;
	HMIWrapping1PistonEnd: STRING;
	HMIWrapping1Piston: STRING;
	bAWrapping1PisHomeRsError: BOOL;
	bAWrapping1PisEndRsError: BOOL;

	TON_Wrapping2PistonOff: BOOL;
	F_TRIG_Wrapping2Piston: F_TRIG;
	bAWrapping2PistonOff: BOOL;
	RS_ErrorWrapping2PistonHome: Rs_Error;
	RS_ErrorWrapping2PistonEnd: Rs_Error;
	HMIWrapping2PistonHome: STRING;
	HMIWrapping2PistonEnd: STRING;
	HMIWrapping2Piston: STRING;
	bAWrapping2PisHomeRsError: BOOL;
	bAWrapping2PisEndRsError: BOOL;
END_VAR
(*......................................Cone Feeding Piston Home Alarm.............................*)

F_TRIG_ConeFeedingPiston(CLK:=bQAConeFeedPisOn , Q=> );

IF F_TRIG_ConeFeedingPiston.Q THEN bAConeFeedingPistonOff:=TRUE;END_IF
IF bIConeFeedingPistonHome THEN bAConeFeedingPistonOff:=FALSE;END_IF



RS_ErrorConeFeedPistonHome(
	bValveOutOn:= bAConeFeedingPistonOff,
	bReedSwithIn:=  bIConeFeedingPistonHome ,
	bErroReset:= bErrorReset ,
	sMsgIn:= ,
	RS_ErrChkDly:=t#5s ,
	bRsError=>bAConeFeedingPistonHomeRsError ,
	sMsgOut=> );

IF RS_ErrorConeFeedPistonHome.bRsError THEN
RS_ErrorConeFeedPistonHome.sMsgIn:='Cone Feeding Piston Home Sensor Timeout Error' ;
ELSE
RS_ErrorConeFeedPistonHome.sMsgIn:='Continue Machine Operation' ;
END_IF
HMIFeedPistonHome:=RS_ErrorConeFeedPistonHome.sMsgIn;

IF bAConeFeedingPistonHomeRsError THEN HMIFeedPiston:=HMIFeedPistonHome;
ELSIF bAConeFeedingPistonEndRsError THEN  HMIFeedPiston:=HMIFeedPistonEnd;
ELSIF NOT bAConeFeedingPistonHomeRsError AND NOT bAConeFeedingPistonEndRsError THEN
HMIFeedPiston:='Continue Machine Running';END_IF


(*......................................Cone Feeding Piston Alarm.............................*)


RS_ErrorConeFeedPistonEnd(
	bValveOutOn:= bQAConeFeedPisOn,
	bReedSwithIn:=  bIConeFeedingPistonEnd ,
	bErroReset:= bErrorReset ,
	sMsgIn:= ,
	RS_ErrChkDly:=t#10s ,
	bRsError=>bAConeFeedingPistonEndRsError ,
	sMsgOut=> );

IF RS_ErrorConeFeedPistonEnd.bRsError THEN
RS_ErrorConeFeedPistonEnd.sMsgIn:='Cone Feeding Piston End Sensor Timeout Error' ;
ELSE
RS_ErrorConeFeedPistonEnd.sMsgIn:='Continue Machine Operation' ;
END_IF
HMIFeedPistonEnd:=RS_ErrorConeFeedPistonEnd.sMsgIn;


(*......................................Cone Forward Piston Home Alarm.............................*)

F_TRIG_ConeForwardPiston(CLK:=bQAForwardPistonOn , Q=> );

IF F_TRIG_ConeForwardPiston.Q THEN bAConeForwardPistonOff:=TRUE;END_IF
IF bIForwardPistonHome THEN bAConeForwardPistonOff:=FALSE;END_IF



RS_ErrorConeForwardPistonHome(
	bValveOutOn:= bAConeForwardPistonOff,
	bReedSwithIn:=  bIForwardPistonHome ,
	bErroReset:= bErrorReset ,
	sMsgIn:= ,
	RS_ErrChkDly:=t#5s ,
	bRsError=>bAForwardPisHomeRsError ,
	sMsgOut=> );

IF RS_ErrorConeForwardPistonHome.bRsError THEN
RS_ErrorConeForwardPistonHome.sMsgIn:='Cone Forward Piston Home Sensor Timeout Error' ;
ELSE
RS_ErrorConeForwardPistonHome.sMsgIn:='Continue Machine Operation' ;
END_IF
HMIForwardPistonHome:=RS_ErrorConeForwardPistonHome.sMsgIn;

IF bAForwardPisHomeRsError THEN HMIForwardPiston:=HMIForwardPistonHome;
ELSIF bAForwardPisEndRsError THEN  HMIForwardPiston:=HMIForwardPistonEnd;
ELSIF NOT bAForwardPisHomeRsError AND NOT bAForwardPisEndRsError THEN
HMIForwardPiston:='Continue Machine Running';END_IF


(*......................................Cone Forward Piston End Alarm.............................*)


RS_ErrorConeForwardPistonEnd(
	bValveOutOn:= bQAForwardPistonOn,
	bReedSwithIn:=  bIForwardPistonEnd ,
	bErroReset:= bErrorReset ,
	sMsgIn:= ,
	RS_ErrChkDly:=t#10s ,
	bRsError=>bAForwardPisEndRsError ,
	sMsgOut=> );

IF RS_ErrorConeForwardPistonEnd.bRsError THEN
RS_ErrorConeForwardPistonEnd.sMsgIn:='Cone Forward Piston End Sensor Timeout Error' ;
ELSE
RS_ErrorConeForwardPistonEnd.sMsgIn:='Continue Machine Operation' ;
END_IF
HMIForwardPistonEnd:=RS_ErrorConeForwardPistonEnd.sMsgIn;


(*......................................Cone Reverse Piston Home Alarm.............................*)

F_TRIG_ConeReversePiston(CLK:=bQAReversePistonOn , Q=> );

IF F_TRIG_ConeReversePiston.Q THEN bAConeReversePistonOff:=TRUE;END_IF
IF bIReversePistonHome THEN bAConeReversePistonOff:=FALSE;END_IF



RS_ErrorConeReversePistonHome(
	bValveOutOn:= bAConeReversePistonOff,
	bReedSwithIn:=  bIReversePistonHome ,
	bErroReset:= bErrorReset ,
	sMsgIn:= ,
	RS_ErrChkDly:=t#5s ,
	bRsError=>bAReversePisHomeRsError ,
	sMsgOut=> );

IF RS_ErrorConeReversePistonHome.bRsError THEN
RS_ErrorConeReversePistonHome.sMsgIn:='Cone Reverse Piston Home Sensor Timeout Error' ;
ELSE
RS_ErrorConeReversePistonHome.sMsgIn:='Continue Machine Operation' ;
END_IF
HMIReversePistonHome:=RS_ErrorConeReversePistonHome.sMsgIn;

IF bAReversePisHomeRsError THEN HMIReversePiston:=HMIReversePistonHome;
ELSIF bAReversePisEndRsError THEN  HMIReversePiston:=HMIReversePistonEnd;
ELSIF NOT bAReversePisHomeRsError AND NOT bAReversePisEndRsError THEN
HMIReversePiston:='Continue Machine Running';END_IF


(*......................................Cone Reverse Piston End Alarm.............................*)


RS_ErrorConeReversePistonEnd(
	bValveOutOn:= bQAReversePistonOn,
	bReedSwithIn:=  bIReversePistonEnd ,
	bErroReset:= bErrorReset ,
	sMsgIn:= ,
	RS_ErrChkDly:=t#10s ,
	bRsError=>bAReversePisEndRsError ,
	sMsgOut=> );

IF RS_ErrorConeReversePistonEnd.bRsError THEN
RS_ErrorConeReversePistonEnd.sMsgIn:='Cone Reverse Piston End Sensor Timeout Error' ;
ELSE
RS_ErrorConeReversePistonEnd.sMsgIn:='Continue Machine Operation' ;
END_IF
HMIReversePistonEnd:=RS_ErrorConeReversePistonEnd.sMsgIn;




(*......................................Cone Tilting Piston Home Alarm.............................*)

F_TRIG_ConeTiltingPiston(CLK:=bQAReversePistonOn , Q=> );

IF F_TRIG_ConeTiltingPiston.Q THEN bAConeTiltingPistonOff:=TRUE;END_IF
IF bIReversePistonHome THEN bAConeTiltingPistonOff:=FALSE;END_IF



RS_ErrorConeTiltingPistonHome(
	bValveOutOn:= bAConeReversePistonOff,
	bReedSwithIn:=  bIReversePistonHome ,
	bErroReset:= bErrorReset ,
	sMsgIn:= ,
	RS_ErrChkDly:=t#5s ,
	bRsError=>bATiltingPisHomeRsError ,
	sMsgOut=> );

IF RS_ErrorConeTiltingPistonHome.bRsError THEN
RS_ErrorConeTiltingPistonHome.sMsgIn:='Cone Tilting Piston Home Sensor Timeout Error' ;
ELSE
RS_ErrorConeTiltingPistonHome.sMsgIn:='Continue Machine Operation' ;
END_IF
HMITiltingPistonHome:=RS_ErrorConeTiltingPistonHome.sMsgIn;

IF bATiltingPisHomeRsError THEN HMITiltingPiston:=HMITiltingPistonHome;
ELSIF bATiltingPisEndRsError THEN  HMITiltingPiston:=HMITiltingPistonEnd;
ELSIF NOT bATiltingPisHomeRsError AND NOT bATiltingPisEndRsError THEN
HMITiltingPiston:='Continue Machine Running';END_IF


(*......................................Cone Tilting Piston End Alarm.............................*)


RS_ErrorConeTiltingPistonEnd(
	bValveOutOn:= bQAReversePistonOn,
	bReedSwithIn:=  bIReversePistonEnd ,
	bErroReset:= bErrorReset ,
	sMsgIn:= ,
	RS_ErrChkDly:=t#10s ,
	bRsError=>bATiltingPisEndRsError ,
	sMsgOut=> );

IF RS_ErrorConeTiltingPistonEnd.bRsError THEN
RS_ErrorConeTiltingPistonEnd.sMsgIn:='Cone Tilting Piston End Sensor Timeout Error' ;
ELSE
RS_ErrorConeTiltingPistonEnd.sMsgIn:='Continue Machine Operation' ;
END_IF
HMITiltingPistonEnd:=RS_ErrorConeTiltingPistonEnd.sMsgIn;




(*......................................Wrapping1 Piston Home Alarm.............................*)

F_TRIG_Wrapping1Piston(CLK:=bQAReversePistonOn , Q=> );

IF F_TRIG_Wrapping1Piston.Q THEN bAWrapping1PistonOff:=TRUE;END_IF
IF bIReversePistonHome THEN bAWrapping1PistonOff:=FALSE;END_IF



RS_ErrorWrapping1PistonHome(
	bValveOutOn:= bAConeReversePistonOff,
	bReedSwithIn:=  bIReversePistonHome ,
	bErroReset:= bErrorReset ,
	sMsgIn:= ,
	RS_ErrChkDly:=t#5s ,
	bRsError=>bAWrapping1PisHomeRsError ,
	sMsgOut=> );

IF RS_ErrorWrapping1PistonHome.bRsError THEN
RS_ErrorWrapping1PistonHome.sMsgIn:='Cone Wrapping1 Piston Home Sensor Timeout Error' ;
ELSE
RS_ErrorWrapping1PistonHome.sMsgIn:='Continue Machine Operation' ;
END_IF
HMIWrapping1PistonHome:=RS_ErrorWrapping1PistonHome.sMsgIn;

IF bAWrapping1PisHomeRsError THEN HMIWrapping1Piston:=HMIWrapping1PistonHome;
ELSIF bAWrapping1PisEndRsError THEN  HMIWrapping1Piston:=HMIWrapping1PistonEnd;
ELSIF NOT bAWrapping1PisHomeRsError AND NOT bAWrapping1PisEndRsError THEN
HMIWrapping1Piston:='Continue Machine Running';END_IF


(*......................................Cone Wrapping1 Piston End Alarm.............................*)


RS_ErrorWrapping1PistonEnd(
	bValveOutOn:= bQAReversePistonOn,
	bReedSwithIn:=  bIReversePistonEnd ,
	bErroReset:= bErrorReset ,
	sMsgIn:= ,
	RS_ErrChkDly:=t#10s ,
	bRsError=>bAWrapping1PisEndRsError ,
	sMsgOut=> );

IF RS_ErrorWrapping1PistonEnd.bRsError THEN
RS_ErrorWrapping1PistonEnd.sMsgIn:='Cone Wrapping1 Piston End Sensor Timeout Error' ;
ELSE
RS_ErrorWrapping1PistonEnd.sMsgIn:='Continue Machine Operation' ;
END_IF
HMIWrapping1PistonEnd:=RS_ErrorWrapping1PistonEnd.sMsgIn;




(*......................................Wrapping2 Piston Home Alarm.............................*)

F_TRIG_Wrapping2Piston(CLK:=bQAReversePistonOn , Q=> );

IF F_TRIG_Wrapping2Piston.Q THEN bAWrapping2PistonOff:=TRUE;END_IF
IF bIReversePistonHome THEN bAWrapping2PistonOff:=FALSE;END_IF



RS_ErrorWrapping2PistonHome(
	bValveOutOn:= bAConeReversePistonOff,
	bReedSwithIn:=  bIReversePistonHome ,
	bErroReset:= bErrorReset ,
	sMsgIn:= ,
	RS_ErrChkDly:=t#5s ,
	bRsError=>bAWrapping2PisHomeRsError ,
	sMsgOut=> );

IF RS_ErrorWrapping2PistonHome.bRsError THEN
RS_ErrorWrapping2PistonHome.sMsgIn:='Cone Wrapping2 Piston Home Sensor Timeout Error' ;
ELSE
RS_ErrorWrapping2PistonHome.sMsgIn:='Continue Machine Operation' ;
END_IF
HMIWrapping2PistonHome:=RS_ErrorWrapping2PistonHome.sMsgIn;

IF bAWrapping2PisHomeRsError THEN HMIWrapping2Piston:=HMIWrapping2PistonHome;
ELSIF bAWrapping2PisEndRsError THEN  HMIWrapping2Piston:=HMIWrapping2PistonEnd;
ELSIF NOT bAWrapping2PisHomeRsError AND NOT bAWrapping2PisEndRsError THEN
HMIWrapping2Piston:='Continue Machine Running';END_IF


(*......................................Cone Wrapping2 Piston End Alarm.............................*)


RS_ErrorWrapping2PistonEnd(
	bValveOutOn:= bQAReversePistonOn,
	bReedSwithIn:=  bIReversePistonEnd ,
	bErroReset:= bErrorReset ,
	sMsgIn:= ,
	RS_ErrChkDly:=t#10s ,
	bRsError=>bAWrapping2PisEndRsError ,
	sMsgOut=> );

IF RS_ErrorWrapping2PistonEnd.bRsError THEN
RS_ErrorWrapping2PistonEnd.sMsgIn:='Cone Wrapping2 Piston End Sensor Timeout Error' ;
ELSE
RS_ErrorWrapping2PistonEnd.sMsgIn:='Continue Machine Operation' ;
END_IF
HMIWrapping2PistonEnd:=RS_ErrorWrapping2PistonEnd.sMsgIn;
END_PROGRAM

(* POU Rs_Error, ST *)
FUNCTION_BLOCK Rs_Error
VAR_INPUT
	bValveOutOn: BOOL;
	bReedSwithIn: BOOL;
	bErroReset: BOOL;
	sMsgIn: STRING;
	RS_ErrChkDly: TIME;
END_VAR
VAR_OUTPUT
	bRsError: BOOL;
	sMsgOut: STRING;
END_VAR
VAR
	FbStep: INT;
	Timer1: TON;
END_VAR
CASE FbStep OF


	0:	Timer1(IN:=FALSE); FbStep:=FbStep+1;

	1:	IF bValveOutOn THEN FbStep:=FbStep+1; END_IF

	2:	Timer1(IN:=TRUE , PT:=RS_ErrChkDly , Q=> , ET=> );
		IF Timer1.Q THEN FbStep:=FbStep+1;
		ELSIF NOT  Timer1.Q AND bReedSwithIn THEN  FbStep:=0; END_IF

	3:	IF bReedSwithIn THEN  FbStep:=FbStep+1;
		ELSIF NOT bReedSwithIn THEN FbStep:=FbStep+2; END_IF

	4:	IF  NOT bValveOutOn THEN sMsgOut:=sMsgIn;  FbStep:=0; END_IF

	5:	bRsError:=TRUE; FbStep:=FbStep+1;

	6:	IF   bReedSwithIn AND   bErroReset THEN bRsError:=FALSE; sMsgOut:='' ;  FbStep:=0;
		ELSIF   NOT bReedSwithIn AND   bRsError  AND  bErroReset THEN bRsError:=FALSE;   sMsgOut:='' ;   FbStep:=0;
		 END_IF

END_CASE
END_FUNCTION_BLOCK

(* POU Outputs, ST *)
PROGRAM Outputs
VAR


END_VAR
				(*O1-EL2809*)

	bQRetA_RowStopperMotorFwd := bQMRetA_RowStopperMotorFwd OR bQRRetA_RowStopperMotorFwd OR bQARetA_RowStopperMotorFwd;
	bQRetA_RowStopperMotorRev := bQMRetA_RowStopperMotorRev OR bQRRetA_RowStopperMotorRev OR bQARetA_RowStopperMotorRev;
	bQRetB_RowStopperMotorFwd := bQMRetB_RowStopperMotorFwd OR bQRRetB_RowStopperMotorFwd OR bQARetB_RowStopperMotorFwd;
	bQRetB_RowStopperMotorRev := bQMRetB_RowStopperMotorRev OR bQRRetB_RowStopperMotorRev OR bQARetB_RowStopperMotorRev;
	bQSpareOutput1 := bQMSpareOutput1 OR bQRSpareOutput1 OR bQASpareOutput1;
	bQRetA_WeightOk := bQARetA_WeightOk ;
	bQRetA_WeightNOk := bQARetA_WeightNOk ;
	bQRetB_WeightOk := bQARetB_WeightOk ;
	bQRetB_WeightNOk :=bQARetB_WeightNOk;
	bQSpareOutput2 := bQMSpareOutput2 OR  bQRSpareOutput2 OR bQASpareOutput2;
	bQSpareOutput3 := bQMSpareOutput3 OR bQRSpareOutput3 OR bQASpareOutput3;
	bQSpareOutput4 :=bQMSpareOutput4 OR bQRSpareOutput4 OR bQASpareOutput4;
	bQTowerLampRed :=bQATowerLampRed OR bQRTowerLampRed;
	bQTowerLampGreen :=bQATowerLampGreen OR bQRTowerLampGreen;
	bQTowerLampYellow :=bQATowerLampYellow OR bQRTowerLampYellow;
	bQTowerBuzzer :=bQATowerBuzzer OR bQRTowerBuzzer;


			(*O2-EL2809*)

	bQConeFeedingPiston :=bQMConeFeedingPiston OR bQRConeFeedingPiston OR bQMConeFeedingPiston;
	bQForwardPiston :=bQMForwardPiston OR bQRForwardPiston OR bQAForwardPiston;
	bQReversePiston :=bQMReversePiston OR bQRReversePiston OR bQAReversePiston;
	bQTiltingPiston :=(bQMTiltingPiston OR bQRTiltingPiston OR bQATiltingPiston);
	bQWrappingPiston1 :=bQMWrappingPiston1 OR bQRWrappingPiston1 OR bQAWrappingPiston1;
	bQWrappingPiston2 :=bQMWrappingPiston2 OR bQRWrappingPiston2 OR bQAWrappingPiston2;
	bQSealingSeparatorYAxisPiston :=bQMSealingSeparatorYAxisPiston OR bQRSealingSeparatorYAxisPiston OR bQASealingSeparatorYAxisPiston;
	bQSealingTopPiston :=bQMSealingTopPiston OR bQRSealingTopPiston OR bQASealingTopPiston;
	bQSealingBottomPiston :=bQMSealingBottomPiston OR bQRSealingBottomPiston OR bQASealingBottomPiston;
	bQSealingSeparatorXAxisPiston :=bQMSealingSeparatorXAxisPiston OR bQRSealingSeparatorXAxisPiston OR bQASealingSeparatorXAxisPiston;
	bQFilmRollerMotor1 :=bQMFilmRollerMotor1 OR bQAFilmRollerMotor1;
	bQFilmRollerMotor2 :=bQMFilmRollerMotor2 OR bQAFilmRollerMotor2;
	bQConeCountPiston :=bQMConeCountPiston OR bQRConeCountPiston OR bQAConeCountPiston;
	bQFeedingConveyorMotor :=bQMFeedingConveyorMotor OR bQRFeedingConveyorMotor OR bQAFeedingConveyorMotor;
	bQWappingConveyorMotor :=bQMWappingConveyorMotor OR bQRWappingConveyorMotor OR bQAWappingConveyorMotor;
	bQSealingConveyorMotor :=bQMSealingConveyorMotor OR  bQRSealingConveyorMotor OR bQASealingConveyorMotor;



			(*O3-EL2008*)

	bQSpareOutput5 :=bQMSpareOutput5 OR bQRSpareOutput5 OR bQASpareOutput5;
	bQSpareOutput6 :=bQMSpareOutput6 OR bQRSpareOutput6 OR bQASpareOutput6;
	bQSpareOutput7 :=bQMSpareOutput7 OR bQRSpareOutput7 OR bQASpareOutput7;
	bQSpareOutput8 :=bQMSpareOutput8 OR bQRSpareOutput8 OR bQASpareOutput8;
	bQSpareOutput9 :=bQMSpareOutput9 OR bQRSpareOutput9 OR bQASpareOutput9;
	bQSpareOutput10 :=bQMSpareOutput10 OR bQRSpareOutput10 OR bQASpareOutput10;
	bQSpareOutput11 :=bQMSpareOutput11 OR bQRSpareOutput11 OR bQASpareOutput11;
	bQSpareOutput12 :=bQMSpareOutput12 OR bQRSpareOutput12 OR bQASpareOutput12;

			(*O4-EL2809*)

	bQColumnStopperPiston :=bQMColumnStopperPiston OR bQRColumnStopperPiston OR bQAColumnStopperPiston;
	bQColumnReversePiston :=bQMColumnReversePiston OR bQRColumnReversePiston OR bAQColumnReversePiston;
	bQSeparatorplatePiston :=bQMSeparatorplatePiston OR bQRSeparatorplatePiston OR bQRSeparatorplatePiston;
	bQConePusher1Piston :=((bQMConePusher1Piston OR bQRConePusher1Piston OR bQAConePusher1Piston) AND NOT bAConePusher1SafetyError);
	bQConePusher2Piston :=bQMConePusher2Piston OR bQRConePusher2Piston OR bQAConePusher2Piston;
	bQBagPusherForwardPiston :=bQMBagPusherForwardPiston OR bQRBagPusherForwardPiston OR bQABagPusherForwardPiston;
	bQBagPusherReversePiston :=bQMBagPusherReversePiston OR bQRBagPusherReversePiston OR bQABagPusherReversePiston;
	bQBagHolderpiston :=bQMBagHolderpiston OR bQRBagHolderpiston OR bQABagHolderpiston;
	bQBagUp_Down180piston :=bQMBagUp_Down180piston OR bQRBagUp_Down180piston OR bQABagUp_Down180piston;
	bQBagUp_Down50piston :=bQMBagUp_Down50piston OR bQRBagUp_Down50piston OR bQABagUp_Down50piston;
	bQBagTiltingpistonForward :=bQMBagTiltingpistonForward OR bQRBagTiltingpistonForward OR bQABagTiltingpistonForward;
	bQBagTiltingpistonReverse :=bQMBagTiltingpistonReverse OR bQRBagTiltingpistonReverse OR bQABagTiltingpistonReverse;
	bQBagRowHolderpiston :=bQBagRowHolderpiston OR bQBagRowHolderpiston OR bQABagRowHolderpiston;
	bQSpareOutput13 :=bQMSpareOutput13 OR bQRSpareOutput13 OR bQASpareOutput13;
	bQSpareOutput14 :=bQMSpareOutput14 OR bQRSpareOutput14 OR bQASpareOutput14;
	bQSpareOutput15 :=bQMSpareOutput15 OR bQRSpareOutput15 OR bQASpareOutput15;
END_PROGRAM

(* POU FilmRollerMotor, ST *)
PROGRAM FilmRollerMotor
VAR

	F_TRIG_1: F_TRIG;
	F_TRIG_2: F_TRIG;
	F_TRIG_11: BOOL;

END_VAR
bQAFilmRollerMotor1:= ( bQAFilmRollerMotor1OnAuto );

bQAFilmRollerMotor2:= ( bQAFilmRollerMotor2OnAuto );


IF NOT bAutoModeOn AND NOT bIFilmTensionRod1Home THEN
bQMFilmRollerMotor1:=TRUE;
ELSE bQMFilmRollerMotor1:=FALSE;
END_IF


IF NOT bAutoModeOn AND NOT bIFilmTensionRod2Home THEN
bQMFilmRollerMotor2:=TRUE;
ELSE bQMFilmRollerMotor2:=FALSE;
END_IF



IF  bAutoModeOn AND NOT bIFilmTensionRod1Home THEN
bQAFilmRollerMotor1:=TRUE;
ELSE bQAFilmRollerMotor1:=FALSE;
END_IF


IF  bAutoModeOn AND NOT bIFilmTensionRod2Home THEN
bQAFilmRollerMotor2:=TRUE;
ELSE bQAFilmRollerMotor2:=FALSE;
END_IF


F_TRIG_1(CLK:=bIFilmTensionRod1Home , Q=> );
F_TRIG_2(CLK:=bIFilmTensionRod2Home , Q=> );


IF bAWrappingConOn AND F_TRIG_1.Q AND NOT  bIWrappingChanelPiston1End THEN bAFilmLoaded1:=TRUE; END_IF

IF bAWrappingConOn AND F_TRIG_2.Q AND NOT  bIWrappingChanelPiston2End THEN bAFilmLoaded2:=TRUE; END_IF
END_PROGRAM

(* POU DalaLog, ST *)
PROGRAM DalaLog
VAR

	TON_Indo1: TON;
	TON_Indo2: TON;
	TON_Indo3: TON;
	TON_Indo4: TON;

	TON_Newdaydly: TON;
	TON_NEWDAY: TON;

	TON_NewdaydlyError: TON;

	TON_writedly: TON;

	TON_Opendly: TON;

END_VAR
;
END_PROGRAM

(* POU Initialization, ST *)
PROGRAM Initialization
VAR




END_VAR
;
END_PROGRAM

(* POU TowerLamp, ST *)
PROGRAM TowerLamp
VAR
	bQTLRed: BOOL;
	bQATLRed: BOOL;
	bAIntBlinkAuto: BOOL;
	bQBuzzer: BOOL;
	bQABuzzer: BOOL;
	bQTLGreen: BOOL;
	bQATLGreen: BOOL;
	bQATLGreenBlnkAuto: BOOL;
	bQTLAmber: BOOL;
	bQATLAmber: BOOL;
	bAEmergencyPressed: BOOL;
	BlinkTimer_1: TON;
	ERROR_ALERT: BOOL;
	BlinkTimer_2: TON;
	BlinkTimer3: TON;
	BlinkTimer4: TON;
	bQAGreenBlnkAuto: BOOL;
	BlinkTimer5: TON;
	BlinkTimer6: TON;
	bTLBlinkOn: BOOL;
	BlinkTimer1: TON;
	BlinkTimer2: TON;
END_VAR
IF bAutoModeOn
THEN
bQTLRed:=  bQATLRed OR bAIntBlinkAuto;

		bQBuzzer:= bQABuzzer;

		bQTLGreen :=(bQATLGreen OR bAIntBlinkAuto OR bQATLGreenBlnkAuto);

		bQTLAmber:=bQATLAmber OR bAIntBlinkAuto;

IF bIMcStopPb OR Stop_TapHmi
THEN bAEmergencyPressed:=TRUE;
ELSE bAEmergencyPressed:=FALSE;
END_IF


BlinkTimer_1(IN:=(ERROR_ALERT AND NOT BlinkTimer_2.Q) , PT:= t#0.5s, Q=> , ET=> );

BlinkTimer_2(IN:= BlinkTimer_1.Q, PT:=t#1.3s , Q=> , ET=> );


BlinkTimer3(IN:= (bAEmergencyPressed AND NOT BlinkTimer4.Q) , PT:= t#0.5s, Q=> , ET=> );

BlinkTimer4(IN:= BlinkTimer3.Q, PT:=t#1.3s , Q=> , ET=> );




IF bAutoModeOn AND (ERROR_ALERT OR bPauseSeq)  AND NOT  bAEmergencyPressed THEN
 bQATLAmber:=TRUE; bQATLGreen:=FALSE;bQATLRed:=FALSE;  ELSE bQATLAmber:=FALSE;
END_IF

IF bAutoModeOn AND (BlinkTimer_1.Q OR BlinkTimer3.Q)
THEN  bQABuzzer:=TRUE;
ELSE bQABuzzer:=FALSE;
END_IF


IF bAutoModeOn AND bAEmergencyPressed
 THEN bQATLRed:=TRUE;bQATLGreen:=FALSE;bQATLAmber:=FALSE;
END_IF

IF bAutoModeOn AND NOT  bAEmergencyPressed AND NOT ERROR_ALERT AND
bMCStartInAuto AND NOT bAMainIntStarted AND NOT IntAllOver  AND NOT  bPauseSeq THEN
bQAGreenBlnkAuto:=TRUE;bQATLAmber:=FALSE;bQATLRed:=FALSE;
ELSE bQAGreenBlnkAuto:=FALSE;
END_IF



BlinkTimer5(IN:= (bQAGreenBlnkAuto AND NOT BlinkTimer6.Q) , PT:= t#0.5s, Q=> , ET=> );
BlinkTimer6(IN:= BlinkTimer5.Q, PT:=t#1.3s , Q=> , ET=> );

IF bAutoModeOn AND BlinkTimer5.Q
THEN bQATLGreenBlnkAuto:=TRUE;
ELSE bQATLGreenBlnkAuto:=FALSE;
END_IF


IF bAutoModeOn AND bMcStartInAuto AND bAMainIntStarted AND NOT  bPauseSeq
AND NOT ERROR_ALERT  AND NOT  bAEmergencyPressed THEN
bTLBlinkOn:=TRUE; bQATLGreen:=FALSE;bQATLAmber:=FALSE; bQATLRed:=FALSE;
ELSE  bTLBlinkOn:=FALSE;
 END_IF

BlinkTimer1(IN:=(bTLBlinkOn AND NOT BlinkTimer2.Q) , PT:= t#0.5s, Q=> , ET=> );

BlinkTimer2(IN:= BlinkTimer1.Q, PT:=t#1.3s , Q=> , ET=> );

IF bAutoModeOn AND  BlinkTimer1.Q
THEN bAIntBlinkAuto:=TRUE;
 ELSE  bAIntBlinkAuto:=FALSE;
 END_IF


IF  bAutoModeOn AND bMCStartInAuto  AND NOT  bAEmergencyPressed AND NOT  bPauseSeq
AND NOT ERROR_ALERT AND NOT bAMainIntStarted AND IntAllOver THEN
 bQATLGreen :=TRUE;bQATLAmber:=FALSE; bQATLRed:=FALSE;
ELSIF NOT IntAllOver THEN bQATLGreen:=FALSE;
 END_IF

END_IF




IF NOT bIAutoManualSwitch
THEN bQATLAmber:=FALSE;bQATLRed:=FALSE;bQATLGreen:=FALSE;bQABuzzer:=FALSE;bAIntBlinkAuto:=FALSE;
END_IF


IF NOT bIAutoManualSwitch THEN bQTLRed:=FALSE;bQBuzzer:=FALSE;bQTLGreen:=FALSE;
bQTLAmber:=FALSE;bQATLRed:=FALSE;bQABuzzer:=FALSE;bQATLGreen:=FALSE;
bQATLGreenBlnkAuto:=FALSE;bQATLAmber:=FALSE;
bAIntBlinkAuto:=FALSE;END_IF
END_PROGRAM

(* Visualisation AA
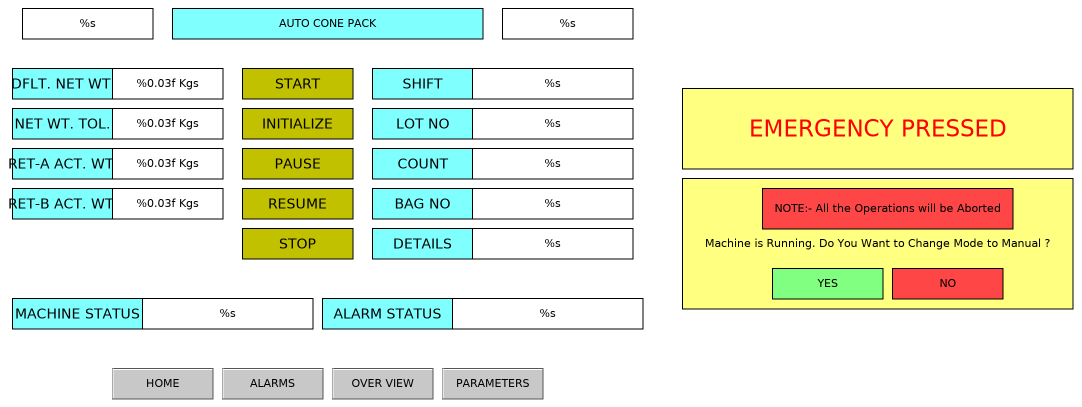
rounded rectangle at (230,80)-(341,111): text "START"; alarm colour if Start_TapHmi; taps Start_TapHmi
rounded rectangle at (230,120)-(341,151): text "INITIALIZE"; alarm colour if Initialize_TapHmi; taps Initialize_TapHmi
rounded rectangle at (230,160)-(341,191): text "PAUSE"; alarm colour if Pause_TapHmi; taps Pause_TapHmi
rounded rectangle at (230,200)-(341,231): text "RESUME"; alarm colour if Resume_TapHmi; taps Resume_TapHmi
rounded rectangle at (230,240)-(341,271): text "STOP"
rectangle at (0,310)-(131,341): text "MACHINE STATUS"
rounded rectangle at (130,310)-(301,341): text "%s"
rectangle at (310,310)-(441,341): text "ALARM STATUS"
rounded rectangle at (440,310)-(631,341): text "%s"
button at (100,380)-(201,411): text "HOME"; opens AA
button at (210,380)-(311,411): text "ALARMS"; opens Alarms
button at (320,380)-(421,411): text "OVER VIEW"; opens Visuvalization
button at (430,380)-(531,411): text "PARAMETERS"; opens Parameters_Load
rectangle at (0,80)-(101,111): text "DFLT. NET WT."
rectangle at (0,120)-(101,151): text "NET WT. TOL."
rectangle at (0,160)-(101,191): text "RET-A ACT. WT."
rectangle at (0,200)-(101,231): text "RET-B ACT. WT."
rounded rectangle at (100,80)-(211,111): text "%0.03f Kgs"
rounded rectangle at (100,120)-(211,151): text "%0.03f Kgs"
rounded rectangle at (100,160)-(211,191): text "%0.03f Kgs"
rounded rectangle at (100,200)-(211,231): text "%0.03f Kgs"
rectangle at (360,80)-(461,111): text "SHIFT"
rectangle at (360,120)-(461,151): text "LOT NO"
rectangle at (360,160)-(461,191): text "COUNT"
rectangle at (360,200)-(461,231): text "BAG NO"
rounded rectangle at (460,80)-(621,111): text "%s"
rectangle at (360,240)-(461,271): text "DETAILS"
rounded rectangle at (460,120)-(621,151): text "%s"
rounded rectangle at (460,160)-(621,191): text "%s"
rounded rectangle at (460,200)-(621,231): text "%s"
rounded rectangle at (460,240)-(621,271): text "%s"
rectangle at (160,20)-(471,51): text "AUTO CONE PACK"
rounded rectangle at (10,20)-(141,51): text "%s"
rounded rectangle at (490,20)-(621,51): text "%s"
rounded rectangle at (670,100)-(1061,181): text "EMERGENCY PRESSED"; invisible if bIEmergencySwitchPb
rounded rectangle at (670,190)-(1061,321): text "Machine is Running. Do You Want to Change Mode to Manual ?"; invisible if NOT bHidePopUp
rounded rectangle at (750,200)-(1001,241): text "NOTE:- All the Operations will be Aborted"; invisible if NOT bHidePopUp
rounded rectangle at (760,280)-(871,311): text "YES"; invisible if NOT bHidePopUp; taps bManualModeOk_TapHmi
rounded rectangle at (880,280)-(991,311): text "NO"; invisible if NOT bHidePopUp; taps bManualModeNOk_TapHmi
*)

(* Visualisation ALARMS
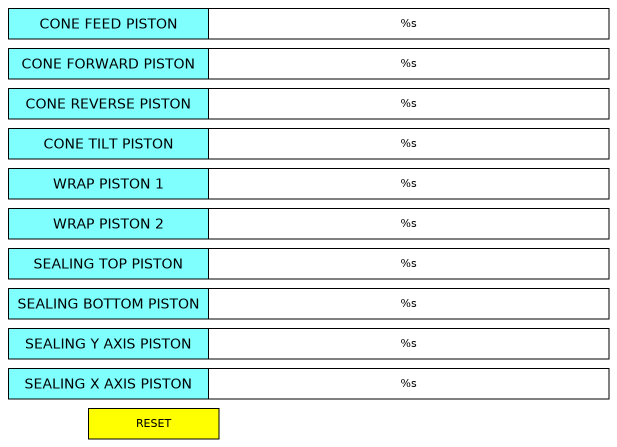
rectangle at (0,40)-(201,71): text "CONE FEED PISTON"
rounded rectangle at (200,40)-(601,71): text "%s"
rectangle at (0,80)-(201,111): text "CONE FORWARD PISTON"
rounded rectangle at (200,80)-(601,111): text "%s"
rectangle at (0,120)-(201,151): text "CONE REVERSE PISTON"
rounded rectangle at (200,120)-(601,151): text "%s"
rectangle at (0,160)-(201,191): text "CONE TILT PISTON"
rounded rectangle at (200,160)-(601,191): text "%s"
rectangle at (0,200)-(201,231): text "WRAP PISTON 1"
rounded rectangle at (200,200)-(601,231): text "%s"
rectangle at (0,240)-(201,271): text "WRAP PISTON 2"
rounded rectangle at (200,240)-(601,271): text "%s"
rectangle at (0,280)-(201,311): text "SEALING TOP PISTON"
rounded rectangle at (200,280)-(601,311): text "%s"
rectangle at (0,320)-(201,351): text "SEALING BOTTOM PISTON"
rounded rectangle at (200,320)-(601,351): text "%s"
rectangle at (0,360)-(201,391): text "SEALING Y AXIS PISTON"
rounded rectangle at (200,360)-(601,391): text "%s"
rectangle at (0,400)-(201,431): text "SEALING X AXIS PISTON"
rounded rectangle at (200,400)-(601,431): text "%s"
rounded rectangle at (80,440)-(211,471): text "RESET"; alarm colour if Reset_TapHmi; taps Reset_TapHmi
*)

(* Visualisation ALARMS_1
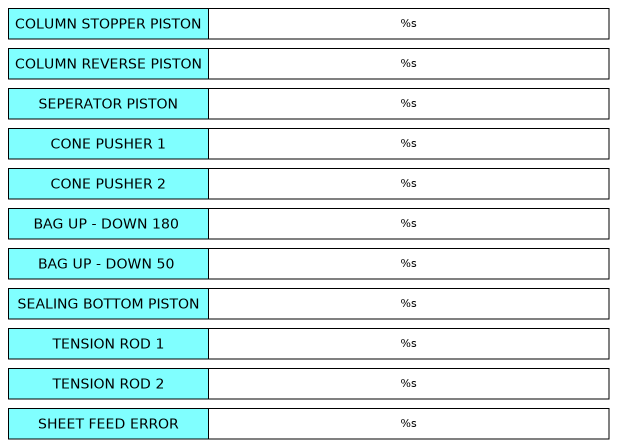
rectangle at (10,10)-(211,41): text "COLUMN STOPPER PISTON"
rounded rectangle at (210,10)-(611,41): text "%s"
rectangle at (10,50)-(211,81): text "COLUMN REVERSE PISTON"
rounded rectangle at (210,50)-(611,81): text "%s"
rectangle at (10,90)-(211,121): text "SEPERATOR PISTON"
rounded rectangle at (210,90)-(611,121): text "%s"
rectangle at (10,130)-(211,161): text "CONE PUSHER 1"
rounded rectangle at (210,130)-(611,161): text "%s"
rectangle at (10,170)-(211,201): text "CONE PUSHER 2"
rounded rectangle at (210,170)-(611,201): text "%s"
rectangle at (10,210)-(211,241): text "BAG UP - DOWN 180"
rounded rectangle at (210,210)-(611,241): text "%s"
rectangle at (10,250)-(211,281): text "BAG UP - DOWN 50"
rounded rectangle at (210,250)-(611,281): text "%s"
rectangle at (10,290)-(211,321): text "SEALING BOTTOM PISTON"
rounded rectangle at (210,290)-(611,321): text "%s"
rectangle at (10,330)-(211,361): text "TENSION ROD 1"
rounded rectangle at (210,330)-(611,361): text "%s"
rectangle at (10,370)-(211,401): text "TENSION ROD 2"
rounded rectangle at (210,370)-(611,401): text "%s"
rectangle at (10,410)-(211,441): text "SHEET FEED ERROR"
rounded rectangle at (210,410)-(611,441): text "%s"
*)

(* Visualisation MANUAL
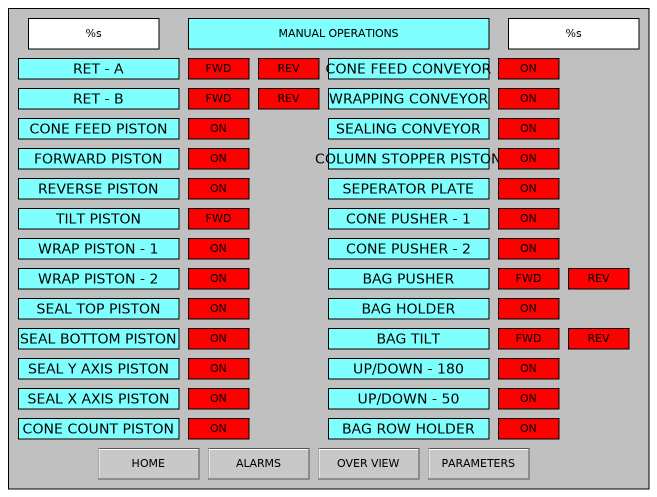
rectangle at (10,50)-(171,71): text "RET - A"
rounded rectangle at (180,50)-(241,71): text "FWD"; alarm colour if bQM_RetA_Fwd; taps bHMI_RetA_Fwd_On
rounded rectangle at (250,50)-(311,71): text "REV"; alarm colour if bQM_RetA_Rev; taps bHMI_Ret_RevA_On
rectangle at (10,80)-(171,101): text "RET - B"
rounded rectangle at (180,80)-(241,101): text "FWD"; alarm colour if bQM_RetB_Fwd; taps bHMI_RetB_Fwd_On
rounded rectangle at (250,80)-(311,101): text "REV"; alarm colour if bQM_RetB_Rev; taps bHMI_Ret_RevB_On
rectangle at (10,110)-(171,131): text "CONE FEED PISTON"
rectangle at (10,140)-(171,161): text "FORWARD PISTON"
rectangle at (10,170)-(171,191): text "REVERSE PISTON"
rectangle at (10,200)-(171,221): text "TILT PISTON"
rectangle at (10,230)-(171,251): text "WRAP PISTON - 1"
rectangle at (10,260)-(171,281): text "WRAP PISTON - 2"
rectangle at (10,290)-(171,311): text "SEAL TOP PISTON"
rectangle at (10,320)-(171,341): text "SEAL BOTTOM PISTON"
rectangle at (10,350)-(171,371): text "SEAL Y AXIS PISTON"
rectangle at (10,380)-(171,401): text "SEAL X AXIS PISTON"
rectangle at (320,50)-(481,71): text "CONE FEED CONVEYOR"
rectangle at (320,80)-(481,101): text "WRAPPING CONVEYOR"
rectangle at (320,110)-(481,131): text "SEALING CONVEYOR"
rectangle at (10,410)-(171,431): text "CONE COUNT PISTON"
rectangle at (320,140)-(481,161): text "COLUMN STOPPER PISTON"
rectangle at (320,170)-(481,191): text "SEPERATOR PLATE"
rectangle at (320,200)-(481,221): text "CONE PUSHER - 1"
rectangle at (320,230)-(481,251): text "CONE PUSHER - 2"
rectangle at (320,260)-(481,281): text "BAG PUSHER"
rectangle at (320,290)-(481,311): text "BAG HOLDER"
rectangle at (320,320)-(481,341): text "BAG TILT"
rectangle at (320,350)-(481,371): text "UP/DOWN - 180"
rectangle at (320,380)-(481,401): text "UP/DOWN - 50"
rectangle at (320,410)-(481,431): text "BAG ROW HOLDER"
rounded rectangle at (180,110)-(241,131): text "ON"; alarm colour if bQM_Cone_Feeding_Piston; toggles bHMI_Cone_Feeding_Piston_On
rounded rectangle at (180,140)-(241,161): text "ON"; alarm colour if bQM_Cone_Forward_Piston; toggles bHMI_Cone_Forward_Piston_On
rounded rectangle at (180,170)-(241,191): text "ON"; alarm colour if bQM_Cone_Reverse_Piston; toggles bHMI_Cone_Reverse_Piston_On
rounded rectangle at (180,200)-(241,221): text "FWD"; alarm colour if bQM_Cone_Tilting_Piston; toggles bHMI_Cone_Tilting_Piston_On
rounded rectangle at (180,230)-(241,251): text "ON"; alarm colour if bQM_Cone_Wrapping_Piston1_Fwd; toggles bHMI_Cone_Wrapping_Piston1_On
rounded rectangle at (180,260)-(241,281): text "ON"; alarm colour if bQM_Cone_Wrapping_Piston2_Fwd; toggles bHMI_Cone_Wrapping_Piston2_On
rounded rectangle at (180,290)-(241,311): text "ON"; alarm colour if bQM_Cone_Sealing_Top_Piston; toggles bHMI_Cone_Sealing_Top_Piston_On
rounded rectangle at (490,260)-(551,281): text "FWD"; alarm colour if bQMBagPusherFwd; taps bIBagPusherFwd_On_Hmi
rounded rectangle at (560,260)-(621,281): text "REV"; alarm colour if bQMBagPusherRev; taps bIBagPusherRev_On_Hmi
button at (90,440)-(191,471): text "HOME"; opens AA
button at (200,440)-(301,471): text "ALARMS"; opens Alarms
button at (310,440)-(411,471): text "OVER VIEW"; opens Visuvalization
button at (420,440)-(521,471): text "PARAMETERS"; opens Parameters_Load
rounded rectangle at (180,10)-(481,41): text "MANUAL OPERATIONS"
rounded rectangle at (180,320)-(241,341): text "ON"; alarm colour if bQM_Cone_Sealing_Bottom_Piston; toggles bHMI_Cone_Sealing_Bottom_Piston_On
rounded rectangle at (180,350)-(241,371): text "ON"; alarm colour if bQM_Cone_Sealing_YAxis_Piston; toggles bHMI_Cone_Sealing_YAxis_Piston_On
rounded rectangle at (180,380)-(241,401): text "ON"; alarm colour if bQM_Cone_Sealing_XAxis_Piston; toggles bHMI_Cone_Sealing_XAxis_Piston_On
rounded rectangle at (180,410)-(241,431): text "ON"; alarm colour if bQM_Cone_Count_Piston; toggles bHMI_Cone_Count_Piston_On
rounded rectangle at (490,50)-(551,71): text "ON"; alarm colour if bQM_Cone_Feeding_Conveyor; toggles bHMI_Cone_Feeding_Conveyor_On
rounded rectangle at (490,80)-(551,101): text "ON"; alarm colour if bQM_Cone_Wrapping_Conveyor; toggles bHMI_Cone_Wrapping_Conveyor_On
rounded rectangle at (490,110)-(551,131): text "ON"; alarm colour if bQM_Cone_Sealing_Conveyor; toggles bHMI_Cone_Sealing_Conveyor_On
rounded rectangle at (490,140)-(551,161): text "ON"; alarm colour if bQMColumnStopperPiston; toggles bIColumn_Stopper_Piston_On_Hmi
rounded rectangle at (490,170)-(551,191): text "ON"; alarm colour if bQMConePusher1; toggles bIConePusher1_On_Hmi
rounded rectangle at (490,200)-(551,221): text "ON"; alarm colour if bQMConePusher2; toggles bIConePusher2_On_Hmi
rounded rectangle at (490,290)-(551,311): text "ON"; alarm colour if bQMBagHolderPiston; toggles bIBagHolder_On_Hmi
rounded rectangle at (490,350)-(551,371): text "ON"; alarm colour if bQMUpDownPiston_1; toggles bIUpDownPiston_1_On_Hmi
rounded rectangle at (490,380)-(551,401): text "ON"; alarm colour if bQMUpDownPiston_2; toggles bIUpDownPiston_2_On_Hmi
rounded rectangle at (490,410)-(551,431): text "ON"; alarm colour if bQMBagRowHolderPiston; toggles bIBagRowHolderPiston_On_Hmi
rounded rectangle at (490,230)-(551,251): text "ON"; alarm colour if bQMConePusher3; toggles bIConePusher3_On_Hmi
rounded rectangle at (490,320)-(551,341): text "FWD"; alarm colour if bQMBagTiltingFwd; taps bIBagTiltingFwd_On_Hmi
rounded rectangle at (560,320)-(621,341): text "REV"; alarm colour if bQMBagTiltingRev; taps bIBagTiltingRev_On_Hmi
rounded rectangle at (20,10)-(151,41): text "%s"
rounded rectangle at (500,10)-(631,41): text "%s"
1 more shapes without text or variables
*)
